LIN {X 0,Y 544.173,Z 839.846,A -85,B 0,C 180,E1 26201.66,E2 26201.66} C_VEL
LIN {X 0,Y 544.039,Z 847.664,A -85,B 0,C 180,E1 26199.734,E2 26199.734} C_VEL
LIN {X 0,Y 543.965,Z 854.535,A -85,B 0,C 180,E1 26197.605,E2 26197.605} C_VEL
LIN {X 0,Y 543.923,Z 859.536,A -85,B 0,C 180,E1 26195.485,E2 26195.485} C_VEL
LIN {X 0,Y 543.91,Z 862.863,A -85,B 0,C 180,E1 26193.445,E2 26193.445} C_VEL
LIN {X 0,Y 543.909,Z 864.729,A -85,B 0,C 180,E1 26191.159,E2 26191.159} C_VEL
LIN {X 0,Y 543.911,Z 864.816,A -85,B 0,C 180,E1 26189.157,E2 26189.157} C_VEL
LIN {X 0,Y 543.916,Z 863.417,A -85,B 0,C 180,E1 26187.05,E2 26187.05} C_VEL
LIN {X 0,Y 543.924,Z 860.152,A -85,B 0,C 180,E1 26184.832,E2 26184.832} C_VEL
LIN {X 0,Y 543.957,Z 855.674,A -85,B 0,C 180,E1 26182.82,E2 26182.82} C_VEL
LIN {X 0,Y 544.034,Z 848.851,A -85,B 0,C 180,E1 26180.586,E2 26180.586} C_VEL
LIN {X 0,Y 544.147,Z 841.239,A -85,B 0,C 180,E1 26178.662,E2 26178.662} C_VEL
LIN {X 0,Y 544.368,Z 831.448,A -85,B 0,C 180,E1 26176.619,E2 26176.619} C_VEL
LIN {X 0,Y 544.661,Z 820.069,A -85,B 0,C 180,E1 26174.672,E2 26174.672} C_VEL
LIN {X 0,Y 545.055,Z 807.802,A -85,B 0,C 180,E1 26172.89,E2 26172.89} C_VEL
LIN {X 0,Y 545.578,Z 792.93,A -85,B 0,C 180,E1 26171.073,E2 26171.073} C_VEL
LIN {X 0,Y 546.089,Z 779.11,A -85,B 0,C 180,E1 26169.629,E2 26169.629} C_VEL
LIN {X 0,Y 546.775,Z 762.015,A -85,B 0,C 180,E1 26168.097,E2 26168.097} C_VEL
LIN {X 0,Y 547.398,Z 745.705,A -85,B 0,C 180,E1 26166.877,E2 26166.877} C_VEL
LIN {X 0,Y 548.047,Z 728.308,A -85,B 0,C 180,E1 26165.765,E2 26165.765} C_VEL
LIN {X 0,Y 548.709,Z 708.264,A -85,B 0,C 180,E1 26164.73,E2 26164.73} C_VEL
LIN {X 0,Y 549.24,Z 690.742,A -85,B 0,C 180,E1 26164.006,E2 26164.006} C_VEL
LIN {X 0,Y 549.747,Z 670.512,A -85,B 0,C 180,E1 26163.357,E2 26163.357} C_VEL
LIN {X 0,Y 550.098,Z 650.393,A -85,B 0,C 180,E1 26162.921,E2 26162.921} C_VEL
LIN {X 0,Y 551.713,Z 417.884,A -85,B 0,C 180,E1 26159.601,E2 26159.601} C_VEL
LIN {X 0,Y 551.587,Z 408.026,A -85,B 0,C 180,E1 26159.447,E2 26159.447} C_VEL
LIN {X 0,Y 547.959,Z 394.771,A -85,B 0,C 180,E1 26158.998,E2 26158.998} C_VEL
LIN {X 0,Y 548.573,Z 372.146,A -85,B 0,C 180,E1 26156.171,E2 26156.171} C_VEL
LIN {X 0,Y 544.361,Z 357.302,A -85,B 0,C 180,E1 26153.906,E2 26153.906} C_VEL
LIN {X 0,Y 544.33,Z 357.175,A -85,B 0,C 180,E1 26150.489,E2 26150.489} C_VEL
LIN {X 0,Y 544.394,Z 357.168,A -85,B 0,C 180,E1 26147.281,E2 26147.281} C_VEL
LIN {X 0,Y 544.328,Z 357.176,A -85,B 0,C 180,E1 26144.094,E2 26144.094} C_VEL
LIN {X 0,Y 544.368,Z 357.177,A -85,B 0,C 180,E1 26140.825,E2 26140.825} C_VEL
LIN {X 0,Y 544.337,Z 357.171,A -85,B 0,C 180,E1 26137.713,E2 26137.713} C_VEL
LIN {X 0,Y 544.334,Z 357.172,A -85,B 0,C 180,E1 26134.329,E2 26134.329} C_VEL
LIN {X 0,Y 544.39,Z 357.175,A -85,B 0,C 180,E1 26131.074,E2 26131.074} C_VEL
LIN {X 0,Y 544.325,Z 357.163,A -85,B 0,C 180,E1 26127.815,E2 26127.815} C_VEL
LIN {X 0,Y 544.364,Z 357.176,A -85,B 0,C 180,E1 26124.529,E2 26124.529} C_VEL
LIN {X 0,Y 544.335,Z 357.165,A -85,B 0,C 180,E1 26121.444,E2 26121.444} C_VEL
LIN {X 0,Y 544.334,Z 357.177,A -85,B 0,C 180,E1 26118.088,E2 26118.088} C_VEL
LIN {X 0,Y 544.378,Z 357.166,A -85,B 0,C 180,E1 26114.904,E2 26114.904} C_VEL
LIN {X 0,Y 544.324,Z 357.175,A -85,B 0,C 180,E1 26111.661,E2 26111.661} C_VEL
LIN {X 0,Y 544.385,Z 357.169,A -85,B 0,C 180,E1 26108.453,E2 26108.453} C_VEL
LIN {X 0,Y 544.329,Z 357.166,A -85,B 0,C 180,E1 26105.274,E2 26105.274} C_VEL
LIN {X 0,Y 544.331,Z 357.176,A -85,B 0,C 180,E1 26101.794,E2 26101.794} C_VEL
LIN {X 0,Y 544.362,Z 357.164,A -85,B 0,C 180,E1 26098.742,E2 26098.742} C_VEL
LIN {X 0,Y 544.324,Z 357.175,A -85,B 0,C 180,E1 26095.475,E2 26095.475} C_VEL
LIN {X 0,Y 544.399,Z 357.166,A -85,B 0,C 180,E1 26092.3,E2 26092.3} C_VEL
LIN {X 0,Y 544.324,Z 357.169,A -85,B 0,C 180,E1 26089.099,E2 26089.099} C_VEL
LIN {X 0,Y 544.344,Z 357.175,A -85,B 0,C 180,E1 26085.757,E2 26085.757} C_VEL
LIN {X 0,Y 544.341,Z 357.162,A -85,B 0,C 180,E1 26082.695,E2 26082.695} C_VEL
LIN {X 0,Y 544.326,Z 357.177,A -85,B 0,C 180,E1 26079.355,E2 26079.355} C_VEL
LIN {X 0,Y 544.386,Z 357.164,A -85,B 0,C 180,E1 26076.154,E2 26076.154} C_VEL
LIN {X 0,Y 544.324,Z 357.177,A -85,B 0,C 180,E1 26072.907,E2 26072.907} C_VEL
LIN {X 0,Y 544.364,Z 357.177,A -85,B 0,C 180,E1 26069.669,E2 26069.669} C_VEL
LIN {X 0,Y 544.323,Z 357.177,A -85,B 0,C 180,E1 26069.105,E2 26069.105} C_VEL
LIN {X 0,Y 543.343,Z 357.304,A -85,B 0,C 180,E1 26068.295,E2 26068.295} C_VEL
LIN {X 0,Y 536.873,Z 358.114,A -85,B 0,C 180,E1 26065.958,E2 26065.958} C_VEL
LIN {X 0,Y 536.406,Z 358.167,A -85,B 0,C 180,E1 26065.424,E2 26065.424} C_VEL
LIN {X 0,Y 536.416,Z 358.165,A -85,B 0,C 180,E1 26062.213,E2 26062.213} C_VEL
LIN {X 0,Y 536.385,Z 358.167,A -85,B 0,C 180,E1 26059.003,E2 26059.003} C_VEL
LIN {X 0,Y 536.448,Z 358.166,A -85,B 0,C 180,E1 26055.817,E2 26055.817} C_VEL
LIN {X 0,Y 536.383,Z 358.167,A -85,B 0,C 180,E1 26052.582,E2 26052.582} C_VEL
LIN {X 0,Y 536.421,Z 358.166,A -85,B 0,C 180,E1 26049.325,E2 26049.325} C_VEL
LIN {X 0,Y 536.395,Z 358.167,A -85,B 0,C 180,E1 26046.197,E2 26046.197} C_VEL
LIN {X 0,Y 536.387,Z 358.167,A -85,B 0,C 180,E1 26042.802,E2 26042.802} C_VEL
LIN {X 0,Y 536.446,Z 358.165,A -85,B 0,C 180,E1 26039.598,E2 26039.598} C_VEL
LIN {X 0,Y 536.382,Z 358.167,A -85,B 0,C 180,E1 26036.336,E2 26036.336} C_VEL
LIN {X 0,Y 536.411,Z 358.167,A -85,B 0,C 180,E1 26032.978,E2 26032.978} C_VEL
LIN {X 0,Y 536.4,Z 358.166,A -85,B 0,C 180,E1 26029.831,E2 26029.831} C_VEL
LIN {X 0,Y 536.383,Z 358.168,A -85,B 0,C 180,E1 26026.459,E2 26026.459} C_VEL
LIN {X 0,Y 536.451,Z 358.165,A -85,B 0,C 180,E1 26023.253,E2 26023.253} C_VEL
LIN {X 0,Y 536.381,Z 358.167,A -85,B 0,C 180,E1 26019.983,E2 26019.983} C_VEL
LIN {X 0,Y 536.4,Z 358.168,A -85,B 0,C 180,E1 26016.602,E2 26016.602} C_VEL
LIN {X 0,Y 536.412,Z 358.166,A -85,B 0,C 180,E1 26013.419,E2 26013.419} C_VEL
LIN {X 0,Y 536.379,Z 358.168,A -85,B 0,C 180,E1 26010.107,E2 26010.107} C_VEL
LIN {X 0,Y 536.443,Z 358.168,A -85,B 0,C 180,E1 26006.902,E2 26006.902} C_VEL
LIN {X 0,Y 536.382,Z 358.168,A -85,B 0,C 180,E1 26003.686,E2 26003.686} C_VEL
LIN {X 0,Y 536.391,Z 358.167,A -85,B 0,C 180,E1 26000.234,E2 26000.234} C_VEL
LIN {X 0,Y 536.436,Z 358.166,A -85,B 0,C 180,E1 25996.966,E2 25996.966} C_VEL
LIN {X 0,Y 536.38,Z 358.168,A -85,B 0,C 180,E1 25993.71,E2 25993.71} C_VEL
LIN {X 0,Y 536.423,Z 358.166,A -85,B 0,C 180,E1 25990.397,E2 25990.397} C_VEL
LIN {X 0,Y 536.388,Z 358.167,A -85,B 0,C 180,E1 25987.303,E2 25987.303} C_VEL
LIN {X 0,Y 536.39,Z 358.167,A -85,B 0,C 180,E1 25983.902,E2 25983.902} C_VEL
LIN {X 0,Y 536.437,Z 358.166,A -85,B 0,C 180,E1 25980.71,E2 25980.71} C_VEL
LIN {X 0,Y 536.381,Z 358.167,A -85,B 0,C 180,E1 25977.531,E2 25977.531} C_VEL
LIN {X 0,Y 536.442,Z 358.167,A -85,B 0,C 180,E1 25974.312,E2 25974.312} C_VEL
LIN {X 0,Y 536.388,Z 358.166,A -85,B 0,C 180,E1 25971.085,E2 25971.085} C_VEL
LIN {X 0,Y 536.387,Z 358.167,A -85,B 0,C 180,E1 25967.564,E2 25967.564} C_VEL
LIN {X 0,Y 536.45,Z 358.165,A -85,B 0,C 180,E1 25964.3,E2 25964.3} C_VEL
LIN {X 0,Y 536.382,Z 358.167,A -85,B 0,C 180,E1 25961.139,E2 25961.139} C_VEL
LIN {X 0,Y 536.42,Z 358.165,A -85,B 0,C 180,E1 25957.815,E2 25957.815} C_VEL
LIN {X 0,Y 536.401,Z 358.167,A -85,B 0,C 180,E1 25954.639,E2 25954.639} C_VEL
LIN {X 0,Y 536.389,Z 358.166,A -85,B 0,C 180,E1 25951.329,E2 25951.329} C_VEL
LIN {X 0,Y 536.446,Z 358.166,A -85,B 0,C 180,E1 25948.128,E2 25948.128} C_VEL
LIN {X 0,Y 536.382,Z 358.158,A -85,B 0,C 180,E1 25944.908,E2 25944.908} C_VEL
LIN {X 0,Y 536.433,Z 358.165,A -85,B 0,C 180,E1 25941.651,E2 25941.651} C_VEL
LIN {X 0,Y 536.399,Z 358.162,A -85,B 0,C 180,E1 25938.421,E2 25938.421} C_VEL
LIN {X 0,Y 536.386,Z 358.163,A -85,B 0,C 180,E1 25935.011,E2 25935.011} C_VEL
LIN {X 0,Y 536.449,Z 358.161,A -85,B 0,C 180,E1 25931.825,E2 25931.825} C_VEL
LIN {X 0,Y 536.383,Z 358.153,A -85,B 0,C 180,E1 25928.571,E2 25928.571} C_VEL
LIN {X 0,Y 536.428,Z 358.164,A -85,B 0,C 180,E1 25925.342,E2 25925.342} C_VEL
LIN {X 0,Y 536.4,Z 358.155,A -85,B 0,C 180,E1 25922.132,E2 25922.132} C_VEL
LIN {X 0,Y 536.388,Z 358.164,A -85,B 0,C 180,E1 25918.714,E2 25918.714} C_VEL
LIN {X 0,Y 536.451,Z 358.156,A -85,B 0,C 180,E1 25915.506,E2 25915.506} C_VEL
LIN {X 0,Y 536.385,Z 358.156,A -85,B 0,C 180,E1 25912.283,E2 25912.283} C_VEL
LIN {X 0,Y 536.413,Z 358.163,A -85,B 0,C 180,E1 25908.927,E2 25908.927} C_VEL
LIN {X 0,Y 536.411,Z 358.151,A -85,B 0,C 180,E1 25905.752,E2 25905.752} C_VEL
LIN {X 0,Y 536.388,Z 358.165,A -85,B 0,C 180,E1 25902.42,E2 25902.42} C_VEL
LIN {X 0,Y 536.455,Z 358.149,A -85,B 0,C 180,E1 25899.142,E2 25899.142} C_VEL
LIN {X 0,Y 536.391,Z 358.165,A -85,B 0,C 180,E1 25895.903,E2 25895.903} C_VEL
LIN {X 0,Y 536.399,Z 358.15,A -85,B 0,C 180,E1 25892.463,E2 25892.463} C_VEL
LIN {X 0,Y 536.442,Z 358.165,A -85,B 0,C 180,E1 25889.229,E2 25889.229} C_VEL
LIN {X 0,Y 536.387,Z 358.161,A -85,B 0,C 180,E1 25885.995,E2 25885.995} C_VEL
LIN {X 0,Y 536.438,Z 358.157,A -85,B 0,C 180,E1 25882.714,E2 25882.714} C_VEL
LIN {X 0,Y 536.396,Z 358.167,A -85,B 0,C 180,E1 25879.555,E2 25879.555} C_VEL
LIN {X 0,Y 536.395,Z 358.165,A -85,B 0,C 180,E1 25876.096,E2 25876.096} C_VEL
LIN {X 0,Y 536.453,Z 358.159,A -85,B 0,C 180,E1 25872.865,E2 25872.865} C_VEL
LIN {X 0,Y 536.389,Z 358.161,A -85,B 0,C 180,E1 25869.605,E2 25869.605} C_VEL
LIN {X 0,Y 536.475,Z 358.365,A -85,B 0,C 180,E1 25866.512,E2 25866.512} C_VEL
LIN {X 0,Y 541.121,Z 374.813,A -85,B 0,C 180,E1 25863.975,E2 25863.975} C_VEL
LIN {X 0,Y 540.557,Z 394.905,A -85,B 0,C 180,E1 25861.456,E2 25861.456} C_VEL
LIN {X 0,Y 544.864,Z 411.254,A -85,B 0,C 180,E1 25860.922,E2 25860.922} C_VEL
LIN {X 0,Y 543.047,Z 645.18,A -85,B 0,C 180,E1 25857.554,E2 25857.554} C_VEL
LIN {X 0,Y 542.717,Z 664.023,A -85,B 0,C 180,E1 25857.181,E2 25857.181} C_VEL
LIN {X 0,Y 542.237,Z 682.867,A -85,B 0,C 180,E1 25856.649,E2 25856.649} C_VEL
LIN {X 0,Y 541.576,Z 703.966,A -85,B 0,C 180,E1 25855.829,E2 25855.829} C_VEL
LIN {X 0,Y 540.927,Z 721.195,A -85,B 0,C 180,E1 25854.983,E2 25854.983} C_VEL
LIN {X 0,Y 540.186,Z 739.996,A -85,B 0,C 180,E1 25853.861,E2 25853.861} C_VEL
LIN {X 0,Y 539.423,Z 757.066,A -85,B 0,C 180,E1 25852.618,E2 25852.618} C_VEL
LIN {X 0,Y 538.693,Z 773.48,A -85,B 0,C 180,E1 25851.218,E2 25851.218} C_VEL
LIN {X 0,Y 537.963,Z 789.942,A -85,B 0,C 180,E1 25849.544,E2 25849.544} C_VEL
LIN {X 0,Y 537.382,Z 803.934,A -85,B 0,C 180,E1 25847.878,E2 25847.878} C_VEL
LIN {X 0,Y 536.859,Z 817.974,A -85,B 0,C 180,E1 25845.889,E2 25845.889} C_VEL
LIN {X 0,Y 536.503,Z 829.096,A -85,B 0,C 180,E1 25844.02,E2 25844.02} C_VEL
LIN {X 0,Y 536.212,Z 839.843,A -85,B 0,C 180,E1 25841.836,E2 25841.836} C_VEL
LIN {X 0,Y 536.058,Z 847.659,A -85,B 0,C 180,E1 25839.88,E2 25839.88} C_VEL
LIN {X 0,Y 535.974,Z 854.538,A -85,B 0,C 180,E1 25837.719,E2 25837.719} C_VEL
LIN {X 0,Y 535.926,Z 859.534,A -85,B 0,C 180,E1 25835.567,E2 25835.567} C_VEL
LIN {X 0,Y 535.91,Z 862.897,A -85,B 0,C 180,E1 25833.468,E2 25833.468} C_VEL
LIN {X 0,Y 535.908,Z 864.725,A -85,B 0,C 180,E1 25831.176,E2 25831.176} C_VEL
LIN {X 0,Y 535.911,Z 864.812,A -85,B 0,C 180,E1 25829.145,E2 25829.145} C_VEL
LIN {X 0,Y 535.915,Z 863.42,A -85,B 0,C 180,E1 25827.006,E2 25827.006} C_VEL
LIN {X 0,Y 535.924,Z 860.15,A -85,B 0,C 180,E1 25824.755,E2 25824.755} C_VEL
LIN {X 0,Y 535.962,Z 855.669,A -85,B 0,C 180,E1 25822.712,E2 25822.712} C_VEL
LIN {X 0,Y 536.051,Z 848.846,A -85,B 0,C 180,E1 25820.445,E2 25820.445} C_VEL
LIN {X 0,Y 536.187,Z 841.236,A -85,B 0,C 180,E1 25818.491,E2 25818.491} C_VEL
LIN {X 0,Y 536.444,Z 831.453,A -85,B 0,C 180,E1 25816.418,E2 25816.418} C_VEL
LIN {X 0,Y 536.784,Z 820.064,A -85,B 0,C 180,E1 25814.442,E2 25814.442} C_VEL
LIN {X 0,Y 537.226,Z 808.102,A -85,B 0,C 180,E1 25812.676,E2 25812.676} C_VEL
LIN {X 0,Y 537.833,Z 793.069,A -85,B 0,C 180,E1 25810.806,E2 25810.806} C_VEL
LIN {X 0,Y 538.42,Z 779.248,A -85,B 0,C 180,E1 25809.34,E2 25809.34} C_VEL
LIN {X 0,Y 539.205,Z 762.007,A -85,B 0,C 180,E1 25807.773,E2 25807.773} C_VEL
LIN {X 0,Y 539.916,Z 745.7,A -85,B 0,C 180,E1 25806.538,E2 25806.538} C_VEL
LIN {X 0,Y 540.61,Z 729.214,A -85,B 0,C 180,E1 25805.468,E2 25805.468} C_VEL
LIN {X 0,Y 541.383,Z 708.932,A -85,B 0,C 180,E1 25804.396,E2 25804.396} C_VEL
LIN {X 0,Y 541.969,Z 691.817,A -85,B 0,C 180,E1 25803.674,E2 25803.674} C_VEL
LIN {X 0,Y 542.539,Z 672.217,A -85,B 0,C 180,E1 25803.023,E2 25803.023} C_VEL
LIN {X 0,Y 542.957,Z 651.512,A -85,B 0,C 180,E1 25802.556,E2 25802.556} C_VEL
LIN {X 0,Y 544.781,Z 422.259,A -85,B 0,C 180,E1 25799.238,E2 25799.238} C_VEL
LIN {X 0,Y 544.663,Z 409.644,A -85,B 0,C 180,E1 25799.041,E2 25799.041} C_VEL
LIN {X 0,Y 540.517,Z 394.526,A -85,B 0,C 180,E1 25798.516,E2 25798.516} C_VEL
LIN {X 0,Y 541.014,Z 374.271,A -85,B 0,C 180,E1 25795.947,E2 25795.947} C_VEL
LIN {X 0,Y 536.462,Z 358.25,A -85,B 0,C 180,E1 25793.448,E2 25793.448} C_VEL
LIN {X 0,Y 536.388,Z 358.156,A -85,B 0,C 180,E1 25790.176,E2 25790.176} C_VEL
LIN {X 0,Y 536.421,Z 358.169,A -85,B 0,C 180,E1 25786.839,E2 25786.839} C_VEL
LIN {X 0,Y 536.415,Z 358.164,A -85,B 0,C 180,E1 25783.606,E2 25783.606} C_VEL
LIN {X 0,Y 536.391,Z 358.167,A -85,B 0,C 180,E1 25780.305,E2 25780.305} C_VEL
LIN {X 0,Y 536.456,Z 358.157,A -85,B 0,C 180,E1 25777.09,E2 25777.09} C_VEL
LIN {X 0,Y 536.39,Z 358.16,A -85,B 0,C 180,E1 25773.876,E2 25773.876} C_VEL
LIN {X 0,Y 536.417,Z 358.165,A -85,B 0,C 180,E1 25770.557,E2 25770.557} C_VEL
LIN {X 0,Y 536.407,Z 358.15,A -85,B 0,C 180,E1 25767.416,E2 25767.416} C_VEL
LIN {X 0,Y 536.389,Z 358.165,A -85,B 0,C 180,E1 25764.026,E2 25764.026} C_VEL
LIN {X 0,Y 536.455,Z 358.149,A -85,B 0,C 180,E1 25760.858,E2 25760.858} C_VEL
LIN {X 0,Y 536.388,Z 358.165,A -85,B 0,C 180,E1 25757.58,E2 25757.58} C_VEL
LIN {X 0,Y 536.411,Z 358.151,A -85,B 0,C 180,E1 25754.247,E2 25754.247} C_VEL
LIN {X 0,Y 536.413,Z 358.163,A -85,B 0,C 180,E1 25751.073,E2 25751.073} C_VEL
LIN {X 0,Y 536.385,Z 358.156,A -85,B 0,C 180,E1 25747.717,E2 25747.717} C_VEL
LIN {X 0,Y 536.451,Z 358.156,A -85,B 0,C 180,E1 25744.494,E2 25744.494} C_VEL
LIN {X 0,Y 536.388,Z 358.164,A -85,B 0,C 180,E1 25741.286,E2 25741.286} C_VEL
LIN {X 0,Y 536.4,Z 358.155,A -85,B 0,C 180,E1 25737.868,E2 25737.868} C_VEL
LIN {X 0,Y 536.428,Z 358.164,A -85,B 0,C 180,E1 25734.658,E2 25734.658} C_VEL
LIN {X 0,Y 536.383,Z 358.153,A -85,B 0,C 180,E1 25731.429,E2 25731.429} C_VEL
LIN {X 0,Y 536.449,Z 358.161,A -85,B 0,C 180,E1 25728.175,E2 25728.175} C_VEL
LIN {X 0,Y 536.386,Z 358.163,A -85,B 0,C 180,E1 25724.989,E2 25724.989} C_VEL
LIN {X 0,Y 536.395,Z 358.162,A -85,B 0,C 180,E1 25721.532,E2 25721.532} C_VEL
LIN {X 0,Y 536.433,Z 358.165,A -85,B 0,C 180,E1 25718.349,E2 25718.349} C_VEL
LIN {X 0,Y 536.382,Z 358.158,A -85,B 0,C 180,E1 25715.092,E2 25715.092} C_VEL
LIN {X 0,Y 536.441,Z 358.166,A -85,B 0,C 180,E1 25711.834,E2 25711.834} C_VEL
LIN {X 0,Y 536.389,Z 358.166,A -85,B 0,C 180,E1 25708.671,E2 25708.671} C_VEL
LIN {X 0,Y 536.406,Z 358.167,A -85,B 0,C 180,E1 25705.424,E2 25705.424} C_VEL
LIN {X 0,Y 535.4,Z 358.29,A -85,B 0,C 180,E1 25704.602,E2 25704.602} C_VEL
LIN {X 0,Y 528.983,Z 359.1,A -85,B 0,C 180,E1 25702.231,E2 25702.231} C_VEL
LIN {X 0,Y 528.504,Z 359.154,A -85,B 0,C 180,E1 25701.689,E2 25701.689} C_VEL
LIN {X 0,Y 528.449,Z 359.155,A -85,B 0,C 180,E1 25698.524,E2 25698.524} C_VEL
LIN {X 0,Y 528.451,Z 359.156,A -85,B 0,C 180,E1 25695.041,E2 25695.041} C_VEL
LIN {X 0,Y 528.51,Z 359.154,A -85,B 0,C 180,E1 25691.752,E2 25691.752} C_VEL
LIN {X 0,Y 528.445,Z 359.155,A -85,B 0,C 180,E1 25688.447,E2 25688.447} C_VEL
LIN {X 0,Y 528.456,Z 359.156,A -85,B 0,C 180,E1 25684.979,E2 25684.979} C_VEL
LIN {X 0,Y 528.493,Z 359.155,A -85,B 0,C 180,E1 25681.731,E2 25681.731} C_VEL
LIN {X 0,Y 528.444,Z 359.155,A -85,B 0,C 180,E1 25678.476,E2 25678.476} C_VEL
LIN {X 0,Y 528.493,Z 359.156,A -85,B 0,C 180,E1 25675.193,E2 25675.193} C_VEL
LIN {X 0,Y 528.451,Z 359.156,A -85,B 0,C 180,E1 25672.001,E2 25672.001} C_VEL
LIN {X 0,Y 528.446,Z 359.156,A -85,B 0,C 180,E1 25668.533,E2 25668.533} C_VEL
LIN {X 0,Y 528.515,Z 359.153,A -85,B 0,C 180,E1 25665.246,E2 25665.246} C_VEL
LIN {X 0,Y 528.443,Z 359.155,A -85,B 0,C 180,E1 25662.012,E2 25662.012} C_VEL
LIN {X 0,Y 528.458,Z 359.157,A -85,B 0,C 180,E1 25658.596,E2 25658.596} C_VEL
LIN {X 0,Y 528.476,Z 359.156,A -85,B 0,C 180,E1 25655.428,E2 25655.428} C_VEL
LIN {X 0,Y 528.439,Z 359.157,A -85,B 0,C 180,E1 25652.06,E2 25652.06} C_VEL
LIN {X 0,Y 528.495,Z 359.157,A -85,B 0,C 180,E1 25648.808,E2 25648.808} C_VEL
LIN {X 0,Y 528.453,Z 359.155,A -85,B 0,C 180,E1 25645.527,E2 25645.527} C_VEL
LIN {X 0,Y 528.448,Z 359.157,A -85,B 0,C 180,E1 25642.171,E2 25642.171} C_VEL
LIN {X 0,Y 528.497,Z 359.155,A -85,B 0,C 180,E1 25638.984,E2 25638.984} C_VEL
LIN {X 0,Y 528.44,Z 359.157,A -85,B 0,C 180,E1 25635.761,E2 25635.761} C_VEL
LIN {X 0,Y 528.485,Z 359.156,A -85,B 0,C 180,E1 25632.436,E2 25632.436} C_VEL
LIN {X 0,Y 528.453,Z 359.155,A -85,B 0,C 180,E1 25629.28,E2 25629.28} C_VEL
LIN {X 0,Y 528.448,Z 359.157,A -85,B 0,C 180,E1 25625.878,E2 25625.878} C_VEL
LIN {X 0,Y 528.516,Z 359.154,A -85,B 0,C 180,E1 25622.513,E2 25622.513} C_VEL
LIN {X 0,Y 528.445,Z 359.156,A -85,B 0,C 180,E1 25619.28,E2 25619.28} C_VEL
LIN {X 0,Y 528.454,Z 359.156,A -85,B 0,C 180,E1 25615.811,E2 25615.811} C_VEL
LIN {X 0,Y 528.492,Z 359.155,A -85,B 0,C 180,E1 25612.604,E2 25612.604} C_VEL
LIN {X 0,Y 528.442,Z 359.155,A -85,B 0,C 180,E1 25609.34,E2 25609.34} C_VEL
LIN {X 0,Y 528.491,Z 359.156,A -85,B 0,C 180,E1 25606.028,E2 25606.028} C_VEL
LIN {X 0,Y 528.461,Z 359.156,A -85,B 0,C 180,E1 25602.77,E2 25602.77} C_VEL
LIN {X 0,Y 528.45,Z 359.155,A -85,B 0,C 180,E1 25599.465,E2 25599.465} C_VEL
LIN {X 0,Y 528.498,Z 359.155,A -85,B 0,C 180,E1 25596.301,E2 25596.301} C_VEL
LIN {X 0,Y 528.445,Z 359.156,A -85,B 0,C 180,E1 25593.011,E2 25593.011} C_VEL
LIN {X 0,Y 528.484,Z 359.155,A -85,B 0,C 180,E1 25589.707,E2 25589.707} C_VEL
LIN {X 0,Y 528.463,Z 359.155,A -85,B 0,C 180,E1 25586.505,E2 25586.505} C_VEL
LIN {X 0,Y 528.449,Z 359.147,A -85,B 0,C 180,E1 25583.145,E2 25583.145} C_VEL
LIN {X 0,Y 528.512,Z 359.153,A -85,B 0,C 180,E1 25579.903,E2 25579.903} C_VEL
LIN {X 0,Y 528.447,Z 359.138,A -85,B 0,C 180,E1 25576.595,E2 25576.595} C_VEL
LIN {X 0,Y 528.456,Z 359.154,A -85,B 0,C 180,E1 25573.117,E2 25573.117} C_VEL
LIN {X 0,Y 528.495,Z 359.138,A -85,B 0,C 180,E1 25569.908,E2 25569.908} C_VEL
LIN {X 0,Y 528.445,Z 359.153,A -85,B 0,C 180,E1 25566.622,E2 25566.622} C_VEL
LIN {X 0,Y 528.492,Z 359.142,A -85,B 0,C 180,E1 25563.357,E2 25563.357} C_VEL
LIN {X 0,Y 528.46,Z 359.143,A -85,B 0,C 180,E1 25560.104,E2 25560.104} C_VEL
LIN {X 0,Y 528.452,Z 359.153,A -85,B 0,C 180,E1 25556.742,E2 25556.742} C_VEL
LIN {X 0,Y 528.516,Z 359.134,A -85,B 0,C 180,E1 25553.478,E2 25553.478} C_VEL
LIN {X 0,Y 528.45,Z 359.154,A -85,B 0,C 180,E1 25550.192,E2 25550.192} C_VEL
LIN {X 0,Y 528.461,Z 359.139,A -85,B 0,C 180,E1 25546.762,E2 25546.762} C_VEL
LIN {X 0,Y 528.482,Z 359.148,A -85,B 0,C 180,E1 25543.623,E2 25543.623} C_VEL
LIN {X 0,Y 528.448,Z 359.149,A -85,B 0,C 180,E1 25540.315,E2 25540.315} C_VEL
LIN {X 0,Y 528.512,Z 359.147,A -85,B 0,C 180,E1 25537.06,E2 25537.06} C_VEL
LIN {X 0,Y 528.455,Z 359.153,A -85,B 0,C 180,E1 25533.839,E2 25533.839} C_VEL
LIN {X 0,Y 528.459,Z 359.153,A -85,B 0,C 180,E1 25530.405,E2 25530.405} C_VEL
LIN {X 0,Y 528.497,Z 359.148,A -85,B 0,C 180,E1 25527.24,E2 25527.24} C_VEL
LIN {X 0,Y 528.449,Z 359.155,A -85,B 0,C 180,E1 25523.951,E2 25523.951} C_VEL
LIN {X 0,Y 528.499,Z 359.155,A -85,B 0,C 180,E1 25520.668,E2 25520.668} C_VEL
LIN {X 0,Y 528.459,Z 359.153,A -85,B 0,C 180,E1 25517.508,E2 25517.508} C_VEL
LIN {X 0,Y 528.455,Z 359.158,A -85,B 0,C 180,E1 25514.028,E2 25514.028} C_VEL
LIN {X 0,Y 528.519,Z 359.123,A -85,B 0,C 180,E1 25510.742,E2 25510.742} C_VEL
LIN {X 0,Y 528.45,Z 359.136,A -85,B 0,C 180,E1 25507.533,E2 25507.533} C_VEL
LIN {X 0,Y 528.547,Z 359.504,A -85,B 0,C 180,E1 25506.943,E2 25506.943} C_VEL
LIN {X 0,Y 533.673,Z 377.481,A -85,B 0,C 180,E1 25504.126,E2 25504.126} C_VEL
LIN {X 0,Y 533.115,Z 394.665,A -85,B 0,C 180,E1 25501.944,E2 25501.944} C_VEL
LIN {X 0,Y 537.976,Z 412.936,A -85,B 0,C 180,E1 25501.334,E2 25501.334} C_VEL
LIN {X 0,Y 535.952,Z 645.248,A -85,B 0,C 180,E1 25497.949,E2 25497.949} C_VEL
LIN {X 0,Y 535.585,Z 663.92,A -85,B 0,C 180,E1 25497.575,E2 25497.575} C_VEL
LIN {X 0,Y 535.084,Z 681.927,A -85,B 0,C 180,E1 25497.064,E2 25497.064} C_VEL
LIN {X 0,Y 534.375,Z 702.71,A -85,B 0,C 180,E1 25496.263,E2 25496.263} C_VEL
LIN {X 0,Y 533.656,Z 719.661,A -85,B 0,C 180,E1 25495.432,E2 25495.432} C_VEL
LIN {X 0,Y 532.875,Z 737.458,A -85,B 0,C 180,E1 25494.38,E2 25494.38} C_VEL
LIN {X 0,Y 531.97,Z 755.622,A -85,B 0,C 180,E1 25493.071,E2 25493.071} C_VEL
LIN {X 0,Y 531.17,Z 771.475,A -85,B 0,C 180,E1 25491.72,E2 25491.72} C_VEL
LIN {X 0,Y 530.317,Z 788.658,A -85,B 0,C 180,E1 25489.986,E2 25489.986} C_VEL
LIN {X 0,Y 529.68,Z 802.156,A -85,B 0,C 180,E1 25488.375,E2 25488.375} C_VEL
LIN {X 0,Y 529.096,Z 815.857,A -85,B 0,C 180,E1 25486.466,E2 25486.466} C_VEL
LIN {X 0,Y 528.65,Z 827.248,A -85,B 0,C 180,E1 25484.569,E2 25484.569} C_VEL
LIN {X 0,Y 528.337,Z 837.389,A -85,B 0,C 180,E1 25482.57,E2 25482.57} C_VEL
LIN {X 0,Y 528.111,Z 846.468,A -85,B 0,C 180,E1 25480.361,E2 25480.361} C_VEL
LIN {X 0,Y 528.002,Z 853.31,A -85,B 0,C 180,E1 25478.274,E2 25478.274} C_VEL
LIN {X 0,Y 527.937,Z 858.915,A -85,B 0,C 180,E1 25475.979,E2 25475.979} C_VEL
LIN {X 0,Y 527.916,Z 862.371,A -85,B 0,C 180,E1 25473.91,E2 25473.91} C_VEL
LIN {X 0,Y 527.907,Z 864.467,A -85,B 0,C 180,E1 25471.737,E2 25471.737} C_VEL
LIN {X 0,Y 527.9,Z 864.895,A -85,B 0,C 180,E1 25469.457,E2 25469.457} C_VEL
LIN {X 0,Y 527.908,Z 863.727,A -85,B 0,C 180,E1 25467.286,E2 25467.286} C_VEL
LIN {X 0,Y 527.928,Z 860.763,A -85,B 0,C 180,E1 25465.002,E2 25465.002} C_VEL
LIN {X 0,Y 527.963,Z 856.429,A -85,B 0,C 180,E1 25462.915,E2 25462.915} C_VEL
LIN {X 0,Y 528.047,Z 850.301,A -85,B 0,C 180,E1 25460.738,E2 25460.738} C_VEL
LIN {X 0,Y 528.208,Z 842.161,A -85,B 0,C 180,E1 25458.536,E2 25458.536} C_VEL
LIN {X 0,Y 528.445,Z 833.662,A -85,B 0,C 180,E1 25456.654,E2 25456.654} C_VEL
LIN {X 0,Y 528.841,Z 822.149,A -85,B 0,C 180,E1 25454.539,E2 25454.539} C_VEL
LIN {X 0,Y 529.302,Z 810.456,A -85,B 0,C 180,E1 25452.749,E2 25452.749} C_VEL
LIN {X 0,Y 529.935,Z 796.797,A -85,B 0,C 180,E1 25450.95,E2 25450.95} C_VEL
LIN {X 0,Y 530.658,Z 781.474,A -85,B 0,C 180,E1 25449.255,E2 25449.255} C_VEL
LIN {X 0,Y 531.462,Z 765.955,A -85,B 0,C 180,E1 25447.782,E2 25447.782} C_VEL
LIN {X 0,Y 532.348,Z 748.104,A -85,B 0,C 180,E1 25446.36,E2 25446.36} C_VEL
LIN {X 0,Y 533.093,Z 731.955,A -85,B 0,C 180,E1 25445.276,E2 25445.276} C_VEL
LIN {X 0,Y 533.967,Z 713.091,A -85,B 0,C 180,E1 25444.218,E2 25444.218} C_VEL
LIN {X 0,Y 534.689,Z 693.683,A -85,B 0,C 180,E1 25443.363,E2 25443.363} C_VEL
LIN {X 0,Y 535.243,Z 676.556,A -85,B 0,C 180,E1 25442.768,E2 25442.768} C_VEL
LIN {X 0,Y 535.797,Z 655.919,A -85,B 0,C 180,E1 25442.239,E2 25442.239} C_VEL
LIN {X 0,Y 536.204,Z 618.298,A -85,B 0,C 180,E1 25441.656,E2 25441.656} C_VEL
LIN {X 0,Y 537.913,Z 411.946,A -85,B 0,C 180,E1 25438.647,E2 25438.647} C_VEL
LIN {X 0,Y 533.079,Z 394.366,A -85,B 0,C 180,E1 25438.036,E2 25438.036} C_VEL
LIN {X 0,Y 533.561,Z 376.939,A -85,B 0,C 180,E1 25435.794,E2 25435.794} C_VEL
LIN {X 0,Y 528.5,Z 359.245,A -85,B 0,C 180,E1 25432.997,E2 25432.997} C_VEL
LIN {X 0,Y 528.465,Z 359.134,A -85,B 0,C 180,E1 25429.823,E2 25429.823} C_VEL
LIN {X 0,Y 528.456,Z 359.158,A -85,B 0,C 180,E1 25426.442,E2 25426.442} C_VEL
LIN {X 0,Y 528.516,Z 359.154,A -85,B 0,C 180,E1 25423.226,E2 25423.226} C_VEL
LIN {X 0,Y 528.452,Z 359.155,A -85,B 0,C 180,E1 25419.981,E2 25419.981} C_VEL
LIN {X 0,Y 528.48,Z 359.156,A -85,B 0,C 180,E1 25416.663,E2 25416.663} C_VEL
LIN {X 0,Y 528.474,Z 359.148,A -85,B 0,C 180,E1 25413.453,E2 25413.453} C_VEL
LIN {X 0,Y 528.451,Z 359.153,A -85,B 0,C 180,E1 25410.095,E2 25410.095} C_VEL
LIN {X 0,Y 528.514,Z 359.14,A -85,B 0,C 180,E1 25406.885,E2 25406.885} C_VEL
LIN {X 0,Y 528.451,Z 359.153,A -85,B 0,C 180,E1 25403.651,E2 25403.651} C_VEL
LIN {X 0,Y 528.462,Z 359.15,A -85,B 0,C 180,E1 25400.214,E2 25400.214} C_VEL
LIN {X 0,Y 528.485,Z 359.154,A -85,B 0,C 180,E1 25397.056,E2 25397.056} C_VEL
LIN {X 0,Y 528.447,Z 359.14,A -85,B 0,C 180,E1 25393.796,E2 25393.796} C_VEL
LIN {X 0,Y 528.502,Z 359.155,A -85,B 0,C 180,E1 25390.468,E2 25390.468} C_VEL
LIN {X 0,Y 528.453,Z 359.144,A -85,B 0,C 180,E1 25387.287,E2 25387.287} C_VEL
LIN {X 0,Y 528.453,Z 359.153,A -85,B 0,C 180,E1 25383.801,E2 25383.801} C_VEL
LIN {X 0,Y 528.52,Z 359.143,A -85,B 0,C 180,E1 25380.438,E2 25380.438} C_VEL
LIN {X 0,Y 528.449,Z 359.143,A -85,B 0,C 180,E1 25377.185,E2 25377.185} C_VEL
LIN {X 0,Y 528.455,Z 359.153,A -85,B 0,C 180,E1 25373.705,E2 25373.705} C_VEL
LIN {X 0,Y 528.493,Z 359.136,A -85,B 0,C 180,E1 25370.532,E2 25370.532} C_VEL
LIN {X 0,Y 528.445,Z 359.155,A -85,B 0,C 180,E1 25367.216,E2 25367.216} C_VEL
LIN {X 0,Y 528.491,Z 359.138,A -85,B 0,C 180,E1 25363.958,E2 25363.958} C_VEL
LIN {X 0,Y 528.463,Z 359.15,A -85,B 0,C 180,E1 25360.671,E2 25360.671} C_VEL
LIN {X 0,Y 528.448,Z 359.147,A -85,B 0,C 180,E1 25357.302,E2 25357.302} C_VEL
LIN {X 0,Y 528.509,Z 359.149,A -85,B 0,C 180,E1 25353.973,E2 25353.973} C_VEL
LIN {X 0,Y 528.45,Z 359.155,A -85,B 0,C 180,E1 25350.717,E2 25350.717} C_VEL
LIN {X 0,Y 528.453,Z 359.156,A -85,B 0,C 180,E1 25347.248,E2 25347.248} C_VEL
LIN {X 0,Y 528.508,Z 359.155,A -85,B 0,C 180,E1 25343.968,E2 25343.968} C_VEL
LIN {X 0,Y 528.504,Z 359.154,A -85,B 0,C 180,E1 25341.689,E2 25341.689} C_VEL
LIN {X 0,Y 527.438,Z 359.283,A -85,B 0,C 180,E1 25340.854,E2 25340.854} C_VEL
LIN {X 0,Y 521.043,Z 360.085,A -85,B 0,C 180,E1 25338.509,E2 25338.509} C_VEL
LIN {X 0,Y 520.565,Z 360.144,A -85,B 0,C 180,E1 25337.898,E2 25337.898} C_VEL
LIN {X 0,Y 520.508,Z 360.145,A -85,B 0,C 180,E1 25334.559,E2 25334.559} C_VEL
LIN {X 0,Y 520.517,Z 360.144,A -85,B 0,C 180,E1 25331.066,E2 25331.066} C_VEL
LIN {X 0,Y 520.548,Z 360.144,A -85,B 0,C 180,E1 25327.88,E2 25327.88} C_VEL
LIN {X 0,Y 520.504,Z 360.145,A -85,B 0,C 180,E1 25324.518,E2 25324.518} C_VEL
LIN {X 0,Y 520.547,Z 360.145,A -85,B 0,C 180,E1 25321.238,E2 25321.238} C_VEL
LIN {X 0,Y 520.516,Z 360.144,A -85,B 0,C 180,E1 25318.074,E2 25318.074} C_VEL
LIN {X 0,Y 520.507,Z 360.146,A -85,B 0,C 180,E1 25314.635,E2 25314.635} C_VEL
LIN {X 0,Y 520.573,Z 360.143,A -85,B 0,C 180,E1 25311.349,E2 25311.349} C_VEL
LIN {X 0,Y 520.509,Z 360.146,A -85,B 0,C 180,E1 25308.015,E2 25308.015} C_VEL
LIN {X 0,Y 520.507,Z 360.146,A -85,B 0,C 180,E1 25304.461,E2 25304.461} C_VEL
LIN {X 0,Y 520.566,Z 360.145,A -85,B 0,C 180,E1 25301.186,E2 25301.186} C_VEL
LIN {X 0,Y 520.503,Z 360.146,A -85,B 0,C 180,E1 25297.95,E2 25297.95} C_VEL
LIN {X 0,Y 520.517,Z 360.145,A -85,B 0,C 180,E1 25294.517,E2 25294.517} C_VEL
LIN {X 0,Y 520.553,Z 360.146,A -85,B 0,C 180,E1 25291.211,E2 25291.211} C_VEL
LIN {X 0,Y 520.501,Z 360.146,A -85,B 0,C 180,E1 25287.908,E2 25287.908} C_VEL
LIN {X 0,Y 520.529,Z 360.146,A -85,B 0,C 180,E1 25284.489,E2 25284.489} C_VEL
LIN {X 0,Y 520.521,Z 360.146,A -85,B 0,C 180,E1 25281.383,E2 25281.383} C_VEL
LIN {X 0,Y 520.506,Z 360.144,A -85,B 0,C 180,E1 25278.027,E2 25278.027} C_VEL
LIN {X 0,Y 520.575,Z 360.142,A -85,B 0,C 180,E1 25274.744,E2 25274.744} C_VEL
LIN {X 0,Y 520.51,Z 360.146,A -85,B 0,C 180,E1 25271.406,E2 25271.406} C_VEL
LIN {X 0,Y 520.509,Z 360.145,A -85,B 0,C 180,E1 25267.884,E2 25267.884} C_VEL
LIN {X 0,Y 520.567,Z 360.143,A -85,B 0,C 180,E1 25264.64,E2 25264.64} C_VEL
LIN {X 0,Y 520.505,Z 360.145,A -85,B 0,C 180,E1 25261.369,E2 25261.369} C_VEL
LIN {X 0,Y 520.526,Z 360.145,A -85,B 0,C 180,E1 25257.985,E2 25257.985} C_VEL
LIN {X 0,Y 520.549,Z 360.145,A -85,B 0,C 180,E1 25254.68,E2 25254.68} C_VEL
LIN {X 0,Y 520.503,Z 360.144,A -85,B 0,C 180,E1 25251.37,E2 25251.37} C_VEL
LIN {X 0,Y 520.549,Z 360.144,A -85,B 0,C 180,E1 25248.056,E2 25248.056} C_VEL
LIN {X 0,Y 520.522,Z 360.145,A -85,B 0,C 180,E1 25244.816,E2 25244.816} C_VEL
LIN {X 0,Y 520.506,Z 360.145,A -85,B 0,C 180,E1 25241.351,E2 25241.351} C_VEL
LIN {X 0,Y 520.57,Z 360.143,A -85,B 0,C 180,E1 25238.051,E2 25238.051} C_VEL
LIN {X 0,Y 520.519,Z 360.145,A -85,B 0,C 180,E1 25234.703,E2 25234.703} C_VEL
LIN {X 0,Y 520.508,Z 360.144,A -85,B 0,C 180,E1 25231.234,E2 25231.234} C_VEL
LIN {X 0,Y 520.576,Z 360.143,A -85,B 0,C 180,E1 25227.934,E2 25227.934} C_VEL
LIN {X 0,Y 520.513,Z 360.135,A -85,B 0,C 180,E1 25224.628,E2 25224.628} C_VEL
LIN {X 0,Y 520.513,Z 360.144,A -85,B 0,C 180,E1 25221.163,E2 25221.163} C_VEL
LIN {X 0,Y 520.571,Z 360.125,A -85,B 0,C 180,E1 25217.891,E2 25217.891} C_VEL
LIN {X 0,Y 520.508,Z 360.141,A -85,B 0,C 180,E1 25214.569,E2 25214.569} C_VEL
LIN {X 0,Y 520.516,Z 360.134,A -85,B 0,C 180,E1 25211.069,E2 25211.069} C_VEL
LIN {X 0,Y 520.58,Z 360.13,A -85,B 0,C 180,E1 25207.679,E2 25207.679} C_VEL
LIN {X 0,Y 520.512,Z 360.142,A -85,B 0,C 180,E1 25204.402,E2 25204.402} C_VEL
LIN {X 0,Y 520.513,Z 360.13,A -85,B 0,C 180,E1 25200.876,E2 25200.876} C_VEL
LIN {X 0,Y 520.561,Z 360.143,A -85,B 0,C 180,E1 25197.684,E2 25197.684} C_VEL
LIN {X 0,Y 520.508,Z 360.13,A -85,B 0,C 180,E1 25194.373,E2 25194.373} C_VEL
LIN {X 0,Y 520.543,Z 360.142,A -85,B 0,C 180,E1 25191.045,E2 25191.045} C_VEL
LIN {X 0,Y 520.533,Z 360.142,A -85,B 0,C 180,E1 25187.798,E2 25187.798} C_VEL
LIN {X 0,Y 520.509,Z 360.136,A -85,B 0,C 180,E1 25184.396,E2 25184.396} C_VEL
LIN {X 0,Y 520.563,Z 360.137,A -85,B 0,C 180,E1 25181.055,E2 25181.055} C_VEL
LIN {X 0,Y 520.522,Z 360.129,A -85,B 0,C 180,E1 25177.761,E2 25177.761} C_VEL
LIN {X 0,Y 520.516,Z 360.141,A -85,B 0,C 180,E1 25174.389,E2 25174.389} C_VEL
LIN {X 0,Y 520.577,Z 360.129,A -85,B 0,C 180,E1 25171.049,E2 25171.049} C_VEL
LIN {X 0,Y 520.514,Z 360.142,A -85,B 0,C 180,E1 25167.85,E2 25167.85} C_VEL
LIN {X 0,Y 520.523,Z 360.144,A -85,B 0,C 180,E1 25164.341,E2 25164.341} C_VEL
LIN {X 0,Y 520.567,Z 360.138,A -85,B 0,C 180,E1 25161.065,E2 25161.065} C_VEL
LIN {X 0,Y 520.513,Z 360.141,A -85,B 0,C 180,E1 25157.751,E2 25157.751} C_VEL
LIN {X 0,Y 520.538,Z 360.146,A -85,B 0,C 180,E1 25154.359,E2 25154.359} C_VEL
LIN {X 0,Y 520.546,Z 360.113,A -85,B 0,C 180,E1 25151.063,E2 25151.063} C_VEL
LIN {X 0,Y 520.511,Z 360.128,A -85,B 0,C 180,E1 25147.789,E2 25147.789} C_VEL
LIN {X 0,Y 520.558,Z 360.422,A -85,B 0,C 180,E1 25147.438,E2 25147.438} C_VEL
LIN {X 0,Y 526.109,Z 379.606,A -85,B 0,C 180,E1 25144.362,E2 25144.362} C_VEL
LIN {X 0,Y 525.724,Z 394.479,A -85,B 0,C 180,E1 25142.442,E2 25142.442} C_VEL
LIN {X 0,Y 531.114,Z 414.653,A -85,B 0,C 180,E1 25141.755,E2 25141.755} C_VEL
LIN {X 0,Y 528.862,Z 646.229,A -85,B 0,C 180,E1 25138.338,E2 25138.338} C_VEL
LIN {X 0,Y 528.475,Z 664.061,A -85,B 0,C 180,E1 25137.974,E2 25137.974} C_VEL
LIN {X 0,Y 527.944,Z 681.558,A -85,B 0,C 180,E1 25137.472,E2 25137.472} C_VEL
LIN {X 0,Y 527.144,Z 702.695,A -85,B 0,C 180,E1 25136.652,E2 25136.652} C_VEL
LIN {X 0,Y 526.384,Z 719.042,A -85,B 0,C 180,E1 25135.844,E2 25135.844} C_VEL
LIN {X 0,Y 525.549,Z 735.614,A -85,B 0,C 180,E1 25134.862,E2 25134.862} C_VEL
LIN {X 0,Y 524.513,Z 754.903,A -85,B 0,C 180,E1 25133.478,E2 25133.478} C_VEL
LIN {X 0,Y 523.662,Z 770.141,A -85,B 0,C 180,E1 25132.172,E2 25132.172} C_VEL
LIN {X 0,Y 522.803,Z 785.906,A -85,B 0,C 180,E1 25130.603,E2 25130.603} C_VEL
LIN {X 0,Y 521.999,Z 800.49,A -85,B 0,C 180,E1 25128.872,E2 25128.872} C_VEL
LIN {X 0,Y 521.381,Z 812.81,A -85,B 0,C 180,E1 25127.177,E2 25127.177} C_VEL
LIN {X 0,Y 520.806,Z 826.013,A -85,B 0,C 180,E1 25125.021,E2 25125.021} C_VEL
LIN {X 0,Y 520.434,Z 835.918,A -85,B 0,C 180,E1 25123.078,E2 25123.078} C_VEL
LIN {X 0,Y 520.164,Z 845.434,A -85,B 0,C 180,E1 25120.81,E2 25120.81} C_VEL
LIN {X 0,Y 520.026,Z 852.314,A -85,B 0,C 180,E1 25118.736,E2 25118.736} C_VEL
LIN {X 0,Y 519.947,Z 857.768,A -85,B 0,C 180,E1 25116.625,E2 25116.625} C_VEL
LIN {X 0,Y 519.911,Z 861.928,A -85,B 0,C 180,E1 25114.301,E2 25114.301} C_VEL
LIN {X 0,Y 519.91,Z 864.245,A -85,B 0,C 180,E1 25112.094,E2 25112.094} C_VEL
LIN {X 0,Y 519.902,Z 864.94,A -85,B 0,C 180,E1 25109.669,E2 25109.669} C_VEL
LIN {X 0,Y 519.902,Z 863.983,A -85,B 0,C 180,E1 25107.575,E2 25107.575} C_VEL
LIN {X 0,Y 519.912,Z 861.624,A -85,B 0,C 180,E1 25105.478,E2 25105.478} C_VEL
LIN {X 0,Y 519.959,Z 857.26,A -85,B 0,C 180,E1 25103.153,E2 25103.153} C_VEL
LIN {X 0,Y 520.035,Z 851.654,A -85,B 0,C 180,E1 25101.041,E2 25101.041} C_VEL
LIN {X 0,Y 520.2,Z 844.007,A -85,B 0,C 180,E1 25098.807,E2 25098.807} C_VEL
LIN {X 0,Y 520.457,Z 835.266,A -85,B 0,C 180,E1 25096.785,E2 25096.785} C_VEL
LIN {X 0,Y 520.861,Z 824.777,A -85,B 0,C 180,E1 25094.753,E2 25094.753} C_VEL
LIN {X 0,Y 521.415,Z 812.023,A -85,B 0,C 180,E1 25092.709,E2 25092.709} C_VEL
LIN {X 0,Y 522.05,Z 799.493,A -85,B 0,C 180,E1 25090.999,E2 25090.999} C_VEL
LIN {X 0,Y 522.902,Z 783.7,A -85,B 0,C 180,E1 25089.167,E2 25089.167} C_VEL
LIN {X 0,Y 523.723,Z 769.083,A -85,B 0,C 180,E1 25087.731,E2 25087.731} C_VEL
LIN {X 0,Y 524.663,Z 752.584,A -85,B 0,C 180,E1 25086.335,E2 25086.335} C_VEL
LIN {X 0,Y 525.605,Z 734.36,A -85,B 0,C 180,E1 25085.058,E2 25085.058} C_VEL
LIN {X 0,Y 526.438,Z 717.982,A -85,B 0,C 180,E1 25084.099,E2 25084.099} C_VEL
LIN {X 0,Y 527.316,Z 698.882,A -85,B 0,C 180,E1 25083.175,E2 25083.175} C_VEL
LIN {X 0,Y 528.005,Z 679.615,A -85,B 0,C 180,E1 25082.466,E2 25082.466} C_VEL
LIN {X 0,Y 528.508,Z 662.583,A -85,B 0,C 180,E1 25081.989,E2 25081.989} C_VEL
LIN {X 0,Y 528.949,Z 641.716,A -85,B 0,C 180,E1 25081.586,E2 25081.586} C_VEL
LIN {X 0,Y 531.104,Z 413.917,A -85,B 0,C 180,E1 25078.233,E2 25078.233} C_VEL
LIN {X 0,Y 525.666,Z 393.926,A -85,B 0,C 180,E1 25077.519,E2 25077.519} C_VEL
LIN {X 0,Y 526.107,Z 379.606,A -85,B 0,C 180,E1 25075.638,E2 25075.638} C_VEL
LIN {X 0,Y 520.534,Z 360.275,A -85,B 0,C 180,E1 25072.532,E2 25072.532} C_VEL
LIN {X 0,Y 520.579,Z 360.109,A -85,B 0,C 180,E1 25069.231,E2 25069.231} C_VEL
LIN {X 0,Y 520.518,Z 360.147,A -85,B 0,C 180,E1 25065.926,E2 25065.926} C_VEL
LIN {X 0,Y 520.517,Z 360.141,A -85,B 0,C 180,E1 25062.397,E2 25062.397} C_VEL
LIN {X 0,Y 520.584,Z 360.138,A -85,B 0,C 180,E1 25059.051,E2 25059.051} C_VEL
LIN {X 0,Y 520.519,Z 360.144,A -85,B 0,C 180,E1 25055.732,E2 25055.732} C_VEL
LIN {X 0,Y 520.518,Z 360.142,A -85,B 0,C 180,E1 25052.28,E2 25052.28} C_VEL
LIN {X 0,Y 520.577,Z 360.129,A -85,B 0,C 180,E1 25048.951,E2 25048.951} C_VEL
LIN {X 0,Y 520.516,Z 360.141,A -85,B 0,C 180,E1 25045.611,E2 25045.611} C_VEL
LIN {X 0,Y 520.516,Z 360.129,A -85,B 0,C 180,E1 25042.12,E2 25042.12} C_VEL
LIN {X 0,Y 520.577,Z 360.139,A -85,B 0,C 180,E1 25038.762,E2 25038.762} C_VEL
LIN {X 0,Y 520.512,Z 360.136,A -85,B 0,C 180,E1 25035.49,E2 25035.49} C_VEL
LIN {X 0,Y 520.517,Z 360.141,A -85,B 0,C 180,E1 25031.977,E2 25031.977} C_VEL
LIN {X 0,Y 520.577,Z 360.135,A -85,B 0,C 180,E1 25028.62,E2 25028.62} C_VEL
LIN {X 0,Y 520.508,Z 360.13,A -85,B 0,C 180,E1 25025.405,E2 25025.405} C_VEL
LIN {X 0,Y 520.528,Z 360.143,A -85,B 0,C 180,E1 25021.986,E2 25021.986} C_VEL
LIN {X 0,Y 520.538,Z 360.126,A -85,B 0,C 180,E1 25018.794,E2 25018.794} C_VEL
LIN {X 0,Y 520.509,Z 360.142,A -85,B 0,C 180,E1 25015.488,E2 25015.488} C_VEL
LIN {X 0,Y 520.563,Z 360.129,A -85,B 0,C 180,E1 25012.167,E2 25012.167} C_VEL
LIN {X 0,Y 520.523,Z 360.134,A -85,B 0,C 180,E1 25008.819,E2 25008.819} C_VEL
LIN {X 0,Y 520.508,Z 360.141,A -85,B 0,C 180,E1 25005.431,E2 25005.431} C_VEL
LIN {X 0,Y 520.571,Z 360.125,A -85,B 0,C 180,E1 25002.109,E2 25002.109} C_VEL
LIN {X 0,Y 520.513,Z 360.144,A -85,B 0,C 180,E1 24998.837,E2 24998.837} C_VEL
LIN {X 0,Y 520.511,Z 360.135,A -85,B 0,C 180,E1 24995.308,E2 24995.308} C_VEL
LIN {X 0,Y 520.572,Z 360.144,A -85,B 0,C 180,E1 24991.936,E2 24991.936} C_VEL
LIN {X 0,Y 520.509,Z 360.144,A -85,B 0,C 180,E1 24988.736,E2 24988.736} C_VEL
LIN {X 0,Y 520.514,Z 360.145,A -85,B 0,C 180,E1 24985.223,E2 24985.223} C_VEL
LIN {X 0,Y 520.571,Z 360.143,A -85,B 0,C 180,E1 24981.945,E2 24981.945} C_VEL
LIN {X 0,Y 520.506,Z 360.145,A -85,B 0,C 180,E1 24978.649,E2 24978.649} C_VEL
LIN {X 0,Y 520.565,Z 360.144,A -85,B 0,C 180,E1 24977.898,E2 24977.898} C_VEL
LIN {X 0,Y 519.732,Z 360.249,A -85,B 0,C 180,E1 24977.11,E2 24977.11} C_VEL
LIN {X 0,Y 515.463,Z 360.779,A -85,B 0,C 180,E1 24975.634,E2 24975.634} C_VEL
LIN {X 0,Y 512.838,Z 361.101,A -85,B 0,C 180,E1 24974.483,E2 24974.483} C_VEL
LIN {X 0,Y 512.603,Z 361.134,A -85,B 0,C 180,E1 24974.047,E2 24974.047} C_VEL
LIN {X 0,Y 512.565,Z 361.133,A -85,B 0,C 180,E1 24970.656,E2 24970.656} C_VEL
LIN {X 0,Y 512.601,Z 361.134,A -85,B 0,C 180,E1 24967.28,E2 24967.28} C_VEL
LIN {X 0,Y 512.589,Z 361.134,A -85,B 0,C 180,E1 24964.018,E2 24964.018} C_VEL
LIN {X 0,Y 512.565,Z 361.134,A -85,B 0,C 180,E1 24960.605,E2 24960.605} C_VEL
LIN {X 0,Y 512.62,Z 361.132,A -85,B 0,C 180,E1 24957.281,E2 24957.281} C_VEL
LIN {X 0,Y 512.581,Z 361.135,A -85,B 0,C 180,E1 24953.936,E2 24953.936} C_VEL
LIN {X 0,Y 512.568,Z 361.133,A -85,B 0,C 180,E1 24950.555,E2 24950.555} C_VEL
LIN {X 0,Y 512.629,Z 361.132,A -85,B 0,C 180,E1 24947.245,E2 24947.245} C_VEL
LIN {X 0,Y 512.568,Z 361.135,A -85,B 0,C 180,E1 24943.997,E2 24943.997} C_VEL
LIN {X 0,Y 512.57,Z 361.135,A -85,B 0,C 180,E1 24940.452,E2 24940.452} C_VEL
LIN {X 0,Y 512.635,Z 361.131,A -85,B 0,C 180,E1 24937.058,E2 24937.058} C_VEL
LIN {X 0,Y 512.573,Z 361.134,A -85,B 0,C 180,E1 24933.691,E2 24933.691} C_VEL
LIN {X 0,Y 512.566,Z 361.136,A -85,B 0,C 180,E1 24930.224,E2 24930.224} C_VEL
LIN {X 0,Y 512.622,Z 361.135,A -85,B 0,C 180,E1 24926.869,E2 24926.869} C_VEL
LIN {X 0,Y 512.576,Z 361.135,A -85,B 0,C 180,E1 24923.504,E2 24923.504} C_VEL
LIN {X 0,Y 512.565,Z 361.135,A -85,B 0,C 180,E1 24920.002,E2 24920.002} C_VEL
LIN {X 0,Y 512.627,Z 361.132,A -85,B 0,C 180,E1 24916.686,E2 24916.686} C_VEL
LIN {X 0,Y 512.571,Z 361.135,A -85,B 0,C 180,E1 24913.454,E2 24913.454} C_VEL
LIN {X 0,Y 512.569,Z 361.133,A -85,B 0,C 180,E1 24909.921,E2 24909.921} C_VEL
LIN {X 0,Y 512.633,Z 361.132,A -85,B 0,C 180,E1 24906.676,E2 24906.676} C_VEL
LIN {X 0,Y 512.571,Z 361.135,A -85,B 0,C 180,E1 24903.286,E2 24903.286} C_VEL
LIN {X 0,Y 512.572,Z 361.133,A -85,B 0,C 180,E1 24899.769,E2 24899.769} C_VEL
LIN {X 0,Y 512.631,Z 361.132,A -85,B 0,C 180,E1 24896.499,E2 24896.499} C_VEL
LIN {X 0,Y 512.568,Z 361.135,A -85,B 0,C 180,E1 24893.213,E2 24893.213} C_VEL
LIN {X 0,Y 512.574,Z 361.133,A -85,B 0,C 180,E1 24889.691,E2 24889.691} C_VEL
LIN {X 0,Y 512.618,Z 361.134,A -85,B 0,C 180,E1 24886.488,E2 24886.488} C_VEL
LIN {X 0,Y 512.567,Z 361.134,A -85,B 0,C 180,E1 24883.153,E2 24883.153} C_VEL
LIN {X 0,Y 512.595,Z 361.133,A -85,B 0,C 180,E1 24879.766,E2 24879.766} C_VEL
LIN {X 0,Y 512.595,Z 361.133,A -85,B 0,C 180,E1 24876.523,E2 24876.523} C_VEL
LIN {X 0,Y 512.57,Z 361.134,A -85,B 0,C 180,E1 24873.195,E2 24873.195} C_VEL
LIN {X 0,Y 512.619,Z 361.133,A -85,B 0,C 180,E1 24869.818,E2 24869.818} C_VEL
LIN {X 0,Y 512.584,Z 361.134,A -85,B 0,C 180,E1 24866.524,E2 24866.524} C_VEL
LIN {X 0,Y 512.57,Z 361.123,A -85,B 0,C 180,E1 24863.077,E2 24863.077} C_VEL
LIN {X 0,Y 512.633,Z 361.128,A -85,B 0,C 180,E1 24859.832,E2 24859.832} C_VEL
LIN {X 0,Y 512.571,Z 361.113,A -85,B 0,C 180,E1 24856.54,E2 24856.54} C_VEL
LIN {X 0,Y 512.572,Z 361.133,A -85,B 0,C 180,E1 24852.957,E2 24852.957} C_VEL
LIN {X 0,Y 512.629,Z 361.108,A -85,B 0,C 180,E1 24849.651,E2 24849.651} C_VEL
LIN {X 0,Y 512.574,Z 361.131,A -85,B 0,C 180,E1 24846.378,E2 24846.378} C_VEL
LIN {X 0,Y 512.575,Z 361.119,A -85,B 0,C 180,E1 24842.902,E2 24842.902} C_VEL
LIN {X 0,Y 512.641,Z 361.119,A -85,B 0,C 180,E1 24839.548,E2 24839.548} C_VEL
LIN {X 0,Y 512.577,Z 361.131,A -85,B 0,C 180,E1 24836.193,E2 24836.193} C_VEL
LIN {X 0,Y 512.576,Z 361.12,A -85,B 0,C 180,E1 24832.711,E2 24832.711} C_VEL
LIN {X 0,Y 512.632,Z 361.133,A -85,B 0,C 180,E1 24829.418,E2 24829.418} C_VEL
LIN {X 0,Y 512.571,Z 361.115,A -85,B 0,C 180,E1 24826.113,E2 24826.113} C_VEL
LIN {X 0,Y 512.581,Z 361.133,A -85,B 0,C 180,E1 24822.632,E2 24822.632} C_VEL
LIN {X 0,Y 512.63,Z 361.113,A -85,B 0,C 180,E1 24819.324,E2 24819.324} C_VEL
LIN {X 0,Y 512.572,Z 361.132,A -85,B 0,C 180,E1 24816.059,E2 24816.059} C_VEL
LIN {X 0,Y 512.602,Z 361.113,A -85,B 0,C 180,E1 24812.714,E2 24812.714} C_VEL
LIN {X 0,Y 512.593,Z 361.132,A -85,B 0,C 180,E1 24809.522,E2 24809.522} C_VEL
LIN {X 0,Y 512.573,Z 361.126,A -85,B 0,C 180,E1 24806.087,E2 24806.087} C_VEL
LIN {X 0,Y 512.621,Z 361.121,A -85,B 0,C 180,E1 24802.728,E2 24802.728} C_VEL
LIN {X 0,Y 512.585,Z 361.134,A -85,B 0,C 180,E1 24799.489,E2 24799.489} C_VEL
LIN {X 0,Y 512.576,Z 361.132,A -85,B 0,C 180,E1 24796.015,E2 24796.015} C_VEL
LIN {X 0,Y 512.631,Z 361.12,A -85,B 0,C 180,E1 24792.663,E2 24792.663} C_VEL
LIN {X 0,Y 512.584,Z 361.124,A -85,B 0,C 180,E1 24789.341,E2 24789.341} C_VEL
LIN {X 0,Y 512.619,Z 361.413,A -85,B 0,C 180,E1 24787.934,E2 24787.934} C_VEL
LIN {X 0,Y 517.769,Z 378.994,A -85,B 0,C 180,E1 24785.035,E2 24785.035} C_VEL
LIN {X 0,Y 518.732,Z 383.694,A -85,B 0,C 180,E1 24784.318,E2 24784.318} C_VEL
LIN {X 0,Y 518.347,Z 394.161,A -85,B 0,C 180,E1 24782.964,E2 24782.964} C_VEL
LIN {X 0,Y 524.28,Z 416.449,A -85,B 0,C 180,E1 24782.187,E2 24782.187} C_VEL
LIN {X 0,Y 521.798,Z 646.608,A -85,B 0,C 180,E1 24778.745,E2 24778.745} C_VEL
LIN {X 0,Y 521.372,Z 664.255,A -85,B 0,C 180,E1 24778.379,E2 24778.379} C_VEL
LIN {X 0,Y 520.776,Z 682.303,A -85,B 0,C 180,E1 24777.852,E2 24777.852} C_VEL
LIN {X 0,Y 519.901,Z 703.163,A -85,B 0,C 180,E1 24777.025,E2 24777.025} C_VEL
LIN {X 0,Y 519.11,Z 718.97,A -85,B 0,C 180,E1 24776.236,E2 24776.236} C_VEL
LIN {X 0,Y 518.22,Z 734.946,A -85,B 0,C 180,E1 24775.282,E2 24775.282} C_VEL
LIN {X 0,Y 517.149,Z 753.476,A -85,B 0,C 180,E1 24773.954,E2 24773.954} C_VEL
LIN {X 0,Y 516.174,Z 769.002,A -85,B 0,C 180,E1 24772.619,E2 24772.619} C_VEL
LIN {X 0,Y 515.283,Z 783.293,A -85,B 0,C 180,E1 24771.199,E2 24771.199} C_VEL
LIN {X 0,Y 514.369,Z 798.6,A -85,B 0,C 180,E1 24769.414,E2 24769.414} C_VEL
LIN {X 0,Y 513.652,Z 811.232,A -85,B 0,C 180,E1 24767.677,E2 24767.677} C_VEL
LIN {X 0,Y 513.046,Z 823.501,A -85,B 0,C 180,E1 24765.717,E2 24765.717} C_VEL
LIN {X 0,Y 512.581,Z 834.187,A -85,B 0,C 180,E1 24763.652,E2 24763.652} C_VEL
LIN {X 0,Y 512.282,Z 842.62,A -85,B 0,C 180,E1 24761.711,E2 24761.711} C_VEL
LIN {X 0,Y 512.071,Z 850.989,A -85,B 0,C 180,E1 24759.326,E2 24759.326} C_VEL
LIN {X 0,Y 511.973,Z 856.722,A -85,B 0,C 180,E1 24757.18,E2 24757.18} C_VEL
LIN {X 0,Y 511.928,Z 861.151,A -85,B 0,C 180,E1 24754.93,E2 24754.93} C_VEL
LIN {X 0,Y 511.908,Z 863.804,A -85,B 0,C 180,E1 24752.687,E2 24752.687} C_VEL
LIN {X 0,Y 511.901,Z 864.888,A -85,B 0,C 180,E1 24750.56,E2 24750.56} C_VEL
LIN {X 0,Y 511.908,Z 864.472,A -85,B 0,C 180,E1 24748.209,E2 24748.209} C_VEL
LIN {X 0,Y 511.916,Z 862.361,A -85,B 0,C 180,E1 24745.968,E2 24745.968} C_VEL
LIN {X 0,Y 511.942,Z 859.116,A -85,B 0,C 180,E1 24743.946,E2 24743.946} C_VEL
LIN {X 0,Y 512.016,Z 853.629,A -85,B 0,C 180,E1 24741.578,E2 24741.578} C_VEL
LIN {X 0,Y 512.163,Z 846.854,A -85,B 0,C 180,E1 24739.426,E2 24739.426} C_VEL
LIN {X 0,Y 512.428,Z 838.428,A -85,B 0,C 180,E1 24737.263,E2 24737.263} C_VEL
LIN {X 0,Y 512.81,Z 828.462,A -85,B 0,C 180,E1 24735.202,E2 24735.202} C_VEL
LIN {X 0,Y 513.308,Z 817.959,A -85,B 0,C 180,E1 24733.362,E2 24733.362} C_VEL
LIN {X 0,Y 514.07,Z 803.909,A -85,B 0,C 180,E1 24731.282,E2 24731.282} C_VEL
LIN {X 0,Y 514.847,Z 790.417,A -85,B 0,C 180,E1 24729.599,E2 24729.599} C_VEL
LIN {X 0,Y 515.836,Z 774.702,A -85,B 0,C 180,E1 24727.912,E2 24727.912} C_VEL
LIN {X 0,Y 516.824,Z 758.506,A -85,B 0,C 180,E1 24726.46,E2 24726.46} C_VEL
LIN {X 0,Y 517.748,Z 743.275,A -85,B 0,C 180,E1 24725.286,E2 24725.286} C_VEL
LIN {X 0,Y 518.839,Z 724.325,A -85,B 0,C 180,E1 24724.059,E2 24724.059} C_VEL
LIN {X 0,Y 519.724,Z 706.706,A -85,B 0,C 180,E1 24723.14,E2 24723.14} C_VEL
LIN {X 0,Y 520.466,Z 689.846,A -85,B 0,C 180,E1 24722.421,E2 24722.421} C_VEL
LIN {X 0,Y 521.257,Z 669.005,A -85,B 0,C 180,E1 24721.74,E2 24721.74} C_VEL
LIN {X 0,Y 521.73,Z 650.102,A -85,B 0,C 180,E1 24721.317,E2 24721.317} C_VEL
LIN {X 0,Y 524.192,Z 424.803,A -85,B 0,C 180,E1 24717.94,E2 24717.94} C_VEL
LIN {X 0,Y 524.081,Z 414.99,A -85,B 0,C 180,E1 24717.777,E2 24717.777} C_VEL
LIN {X 0,Y 518.293,Z 393.711,A -85,B 0,C 180,E1 24717.005,E2 24717.005} C_VEL
LIN {X 0,Y 518.643,Z 382.231,A -85,B 0,C 180,E1 24715.475,E2 24715.475} C_VEL
LIN {X 0,Y 513.233,Z 363.475,A -85,B 0,C 180,E1 24712.428,E2 24712.428} C_VEL
LIN {X 0,Y 512.589,Z 361.191,A -85,B 0,C 180,E1 24712.006,E2 24712.006} C_VEL
LIN {X 0,Y 512.573,Z 361.108,A -85,B 0,C 180,E1 24708.455,E2 24708.455} C_VEL
LIN {X 0,Y 512.632,Z 361.124,A -85,B 0,C 180,E1 24705.087,E2 24705.087} C_VEL
LIN {X 0,Y 512.58,Z 361.128,A -85,B 0,C 180,E1 24701.83,E2 24701.83} C_VEL
LIN {X 0,Y 512.578,Z 361.125,A -85,B 0,C 180,E1 24698.341,E2 24698.341} C_VEL
LIN {X 0,Y 512.637,Z 361.129,A -85,B 0,C 180,E1 24694.992,E2 24694.992} C_VEL
LIN {X 0,Y 512.581,Z 361.131,A -85,B 0,C 180,E1 24691.653,E2 24691.653} C_VEL
LIN {X 0,Y 512.575,Z 361.114,A -85,B 0,C 180,E1 24688.156,E2 24688.156} C_VEL
LIN {X 0,Y 512.634,Z 361.133,A -85,B 0,C 180,E1 24684.797,E2 24684.797} C_VEL
LIN {X 0,Y 512.578,Z 361.116,A -85,B 0,C 180,E1 24681.498,E2 24681.498} C_VEL
LIN {X 0,Y 512.573,Z 361.133,A -85,B 0,C 180,E1 24677.955,E2 24677.955} C_VEL
LIN {X 0,Y 512.629,Z 361.109,A -85,B 0,C 180,E1 24674.577,E2 24674.577} C_VEL
LIN {X 0,Y 512.583,Z 361.13,A -85,B 0,C 180,E1 24671.253,E2 24671.253} C_VEL
LIN {X 0,Y 512.574,Z 361.12,A -85,B 0,C 180,E1 24667.852,E2 24667.852} C_VEL
LIN {X 0,Y 512.632,Z 361.118,A -85,B 0,C 180,E1 24664.591,E2 24664.591} C_VEL
LIN {X 0,Y 512.575,Z 361.131,A -85,B 0,C 180,E1 24661.234,E2 24661.234} C_VEL
LIN {X 0,Y 512.572,Z 361.119,A -85,B 0,C 180,E1 24657.657,E2 24657.657} C_VEL
LIN {X 0,Y 512.634,Z 361.132,A -85,B 0,C 180,E1 24654.297,E2 24654.297} C_VEL
LIN {X 0,Y 512.574,Z 361.116,A -85,B 0,C 180,E1 24651.028,E2 24651.028} C_VEL
LIN {X 0,Y 512.573,Z 361.133,A -85,B 0,C 180,E1 24647.501,E2 24647.501} C_VEL
LIN {X 0,Y 512.634,Z 361.114,A -85,B 0,C 180,E1 24644.16,E2 24644.16} C_VEL
LIN {X 0,Y 512.581,Z 361.127,A -85,B 0,C 180,E1 24640.748,E2 24640.748} C_VEL
LIN {X 0,Y 512.57,Z 361.124,A -85,B 0,C 180,E1 24637.287,E2 24637.287} C_VEL
LIN {X 0,Y 512.629,Z 361.126,A -85,B 0,C 180,E1 24633.977,E2 24633.977} C_VEL
LIN {X 0,Y 512.575,Z 361.133,A -85,B 0,C 180,E1 24630.682,E2 24630.682} C_VEL
LIN {X 0,Y 512.572,Z 361.134,A -85,B 0,C 180,E1 24627.169,E2 24627.169} C_VEL
LIN {X 0,Y 512.628,Z 361.133,A -85,B 0,C 180,E1 24623.782,E2 24623.782} C_VEL
LIN {X 0,Y 512.573,Z 361.133,A -85,B 0,C 180,E1 24620.522,E2 24620.522} C_VEL
LIN {X 0,Y 512.571,Z 361.134,A -85,B 0,C 180,E1 24617.011,E2 24617.011} C_VEL
LIN {X 0,Y 512.603,Z 361.134,A -85,B 0,C 180,E1 24614.047,E2 24614.047} C_VEL
LIN {X 0,Y 511.788,Z 361.24,A -85,B 0,C 180,E1 24613.247,E2 24613.247} C_VEL
LIN {X 0,Y 507.718,Z 361.744,A -85,B 0,C 180,E1 24611.807,E2 24611.807} C_VEL
LIN {X 0,Y 504.972,Z 362.08,A -85,B 0,C 180,E1 24610.641,E2 24610.641} C_VEL
LIN {X 0,Y 504.648,Z 362.122,A -85,B 0,C 180,E1 24610.135,E2 24610.135} C_VEL
LIN {X 0,Y 504.629,Z 362.123,A -85,B 0,C 180,E1 24606.752,E2 24606.752} C_VEL
LIN {X 0,Y 504.687,Z 362.121,A -85,B 0,C 180,E1 24603.418,E2 24603.418} C_VEL
LIN {X 0,Y 504.642,Z 362.123,A -85,B 0,C 180,E1 24600.039,E2 24600.039} C_VEL
LIN {X 0,Y 504.629,Z 362.124,A -85,B 0,C 180,E1 24596.601,E2 24596.601} C_VEL
LIN {X 0,Y 504.682,Z 362.123,A -85,B 0,C 180,E1 24593.204,E2 24593.204} C_VEL
LIN {X 0,Y 504.638,Z 362.122,A -85,B 0,C 180,E1 24589.924,E2 24589.924} C_VEL
LIN {X 0,Y 504.629,Z 362.125,A -85,B 0,C 180,E1 24586.459,E2 24586.459} C_VEL
LIN {X 0,Y 504.691,Z 362.122,A -85,B 0,C 180,E1 24583.169,E2 24583.169} C_VEL
LIN {X 0,Y 504.634,Z 362.124,A -85,B 0,C 180,E1 24579.811,E2 24579.811} C_VEL
LIN {X 0,Y 504.63,Z 362.124,A -85,B 0,C 180,E1 24576.37,E2 24576.37} C_VEL
LIN {X 0,Y 504.683,Z 362.122,A -85,B 0,C 180,E1 24572.953,E2 24572.953} C_VEL
LIN {X 0,Y 504.632,Z 362.125,A -85,B 0,C 180,E1 24569.659,E2 24569.659} C_VEL
LIN {X 0,Y 504.627,Z 362.123,A -85,B 0,C 180,E1 24566.137,E2 24566.137} C_VEL
LIN {X 0,Y 504.694,Z 362.12,A -85,B 0,C 180,E1 24562.83,E2 24562.83} C_VEL
LIN {X 0,Y 504.634,Z 362.124,A -85,B 0,C 180,E1 24559.497,E2 24559.497} C_VEL
LIN {X 0,Y 504.63,Z 362.124,A -85,B 0,C 180,E1 24556.012,E2 24556.012} C_VEL
LIN {X 0,Y 504.69,Z 362.121,A -85,B 0,C 180,E1 24552.698,E2 24552.698} C_VEL
LIN {X 0,Y 504.633,Z 362.122,A -85,B 0,C 180,E1 24549.349,E2 24549.349} C_VEL
LIN {X 0,Y 504.63,Z 362.124,A -85,B 0,C 180,E1 24545.787,E2 24545.787} C_VEL
LIN {X 0,Y 504.682,Z 362.123,A -85,B 0,C 180,E1 24542.382,E2 24542.382} C_VEL
LIN {X 0,Y 504.641,Z 362.123,A -85,B 0,C 180,E1 24539.067,E2 24539.067} C_VEL
LIN {X 0,Y 504.63,Z 362.124,A -85,B 0,C 180,E1 24535.62,E2 24535.62} C_VEL
LIN {X 0,Y 504.681,Z 362.122,A -85,B 0,C 180,E1 24532.218,E2 24532.218} C_VEL
LIN {X 0,Y 504.645,Z 362.122,A -85,B 0,C 180,E1 24528.87,E2 24528.87} C_VEL
LIN {X 0,Y 504.63,Z 362.123,A -85,B 0,C 180,E1 24525.462,E2 24525.462} C_VEL
LIN {X 0,Y 504.695,Z 362.121,A -85,B 0,C 180,E1 24522.18,E2 24522.18} C_VEL
LIN {X 0,Y 504.635,Z 362.122,A -85,B 0,C 180,E1 24518.863,E2 24518.863} C_VEL
LIN {X 0,Y 504.631,Z 362.123,A -85,B 0,C 180,E1 24515.284,E2 24515.284} C_VEL
LIN {X 0,Y 504.688,Z 362.122,A -85,B 0,C 180,E1 24511.927,E2 24511.927} C_VEL
LIN {X 0,Y 504.641,Z 362.122,A -85,B 0,C 180,E1 24508.634,E2 24508.634} C_VEL
LIN {X 0,Y 504.63,Z 362.111,A -85,B 0,C 180,E1 24505.115,E2 24505.115} C_VEL
LIN {X 0,Y 504.681,Z 362.12,A -85,B 0,C 180,E1 24501.699,E2 24501.699} C_VEL
LIN {X 0,Y 504.648,Z 362.114,A -85,B 0,C 180,E1 24498.356,E2 24498.356} C_VEL
LIN {X 0,Y 504.629,Z 362.118,A -85,B 0,C 180,E1 24494.92,E2 24494.92} C_VEL
LIN {X 0,Y 504.689,Z 362.111,A -85,B 0,C 180,E1 24491.652,E2 24491.652} C_VEL
LIN {X 0,Y 504.64,Z 362.104,A -85,B 0,C 180,E1 24488.311,E2 24488.311} C_VEL
LIN {X 0,Y 504.633,Z 362.12,A -85,B 0,C 180,E1 24484.768,E2 24484.768} C_VEL
LIN {X 0,Y 504.676,Z 362.097,A -85,B 0,C 180,E1 24481.357,E2 24481.357} C_VEL
LIN {X 0,Y 504.647,Z 362.12,A -85,B 0,C 180,E1 24478.065,E2 24478.065} C_VEL
LIN {X 0,Y 504.633,Z 362.105,A -85,B 0,C 180,E1 24474.652,E2 24474.652} C_VEL
LIN {X 0,Y 504.694,Z 362.112,A -85,B 0,C 180,E1 24471.32,E2 24471.32} C_VEL
LIN {X 0,Y 504.641,Z 362.119,A -85,B 0,C 180,E1 24467.988,E2 24467.988} C_VEL
LIN {X 0,Y 504.634,Z 362.113,A -85,B 0,C 180,E1 24464.481,E2 24464.481} C_VEL
LIN {X 0,Y 504.693,Z 362.115,A -85,B 0,C 180,E1 24461.156,E2 24461.156} C_VEL
LIN {X 0,Y 504.645,Z 362.105,A -85,B 0,C 180,E1 24457.76,E2 24457.76} C_VEL
LIN {X 0,Y 504.635,Z 362.119,A -85,B 0,C 180,E1 24454.28,E2 24454.28} C_VEL
LIN {X 0,Y 504.686,Z 362.109,A -85,B 0,C 180,E1 24450.887,E2 24450.887} C_VEL
LIN {X 0,Y 504.653,Z 362.119,A -85,B 0,C 180,E1 24447.522,E2 24447.522} C_VEL
LIN {X 0,Y 504.635,Z 362.122,A -85,B 0,C 180,E1 24444.089,E2 24444.089} C_VEL
LIN {X 0,Y 504.693,Z 362.12,A -85,B 0,C 180,E1 24440.768,E2 24440.768} C_VEL
LIN {X 0,Y 504.645,Z 362.119,A -85,B 0,C 180,E1 24437.479,E2 24437.479} C_VEL
LIN {X 0,Y 504.639,Z 362.126,A -85,B 0,C 180,E1 24434.007,E2 24434.007} C_VEL
LIN {X 0,Y 504.694,Z 362.082,A -85,B 0,C 180,E1 24430.642,E2 24430.642} C_VEL
LIN {X 0,Y 504.716,Z 362.382,A -85,B 0,C 180,E1 24428.45,E2 24428.45} C_VEL
LIN {X 0,Y 509.821,Z 379.921,A -85,B 0,C 180,E1 24425.485,E2 24425.485} C_VEL
LIN {X 0,Y 511.302,Z 385.825,A -85,B 0,C 180,E1 24424.547,E2 24424.547} C_VEL
LIN {X 0,Y 511.004,Z 393.904,A -85,B 0,C 180,E1 24423.5,E2 24423.5} C_VEL
LIN {X 0,Y 517.476,Z 418.315,A -85,B 0,C 180,E1 24422.628,E2 24422.628} C_VEL
LIN {X 0,Y 514.758,Z 647.09,A -85,B 0,C 180,E1 24419.162,E2 24419.162} C_VEL
LIN {X 0,Y 514.288,Z 664.641,A -85,B 0,C 180,E1 24418.789,E2 24418.789} C_VEL
LIN {X 0,Y 513.583,Z 684.221,A -85,B 0,C 180,E1 24418.202,E2 24418.202} C_VEL
LIN {X 0,Y 512.657,Z 703.609,A -85,B 0,C 180,E1 24417.404,E2 24417.404} C_VEL
LIN {X 0,Y 511.768,Z 719.845,A -85,B 0,C 180,E1 24416.576,E2 24416.576} C_VEL
LIN {X 0,Y 510.779,Z 736.365,A -85,B 0,C 180,E1 24415.57,E2 24415.57} C_VEL
LIN {X 0,Y 509.603,Z 754.855,A -85,B 0,C 180,E1 24414.208,E2 24414.208} C_VEL
LIN {X 0,Y 508.633,Z 769.063,A -85,B 0,C 180,E1 24412.967,E2 24412.967} C_VEL
LIN {X 0,Y 507.68,Z 783.129,A -85,B 0,C 180,E1 24411.549,E2 24411.549} C_VEL
LIN {X 0,Y 506.654,Z 798.608,A -85,B 0,C 180,E1 24409.72,E2 24409.72} C_VEL
LIN {X 0,Y 505.904,Z 810.453,A -85,B 0,C 180,E1 24408.074,E2 24408.074} C_VEL
LIN {X 0,Y 505.283,Z 821.468,A -85,B 0,C 180,E1 24406.314,E2 24406.314} C_VEL
LIN {X 0,Y 504.711,Z 833.108,A -85,B 0,C 180,E1 24404.103,E2 24404.103} C_VEL
LIN {X 0,Y 504.353,Z 841.688,A -85,B 0,C 180,E1 24402.13,E2 24402.13} C_VEL
LIN {X 0,Y 504.119,Z 849.603,A -85,B 0,C 180,E1 24399.936,E2 24399.936} C_VEL
LIN {X 0,Y 503.99,Z 855.916,A -85,B 0,C 180,E1 24397.638,E2 24397.638} C_VEL
LIN {X 0,Y 503.933,Z 860.142,A -85,B 0,C 180,E1 24395.579,E2 24395.579} C_VEL
LIN {X 0,Y 503.913,Z 863.433,A -85,B 0,C 180,E1 24393.185,E2 24393.185} C_VEL
LIN {X 0,Y 503.912,Z 864.797,A -85,B 0,C 180,E1 24390.909,E2 24390.909} C_VEL
LIN {X 0,Y 503.91,Z 864.739,A -85,B 0,C 180,E1 24388.863,E2 24388.863} C_VEL
LIN {X 0,Y 503.912,Z 863.033,A -85,B 0,C 180,E1 24386.432,E2 24386.432} C_VEL
LIN {X 0,Y 503.936,Z 859.936,A -85,B 0,C 180,E1 24384.307,E2 24384.307} C_VEL
LIN {X 0,Y 503.996,Z 855.649,A -85,B 0,C 180,E1 24382.247,E2 24382.247} C_VEL
LIN {X 0,Y 504.135,Z 848.827,A -85,B 0,C 180,E1 24379.833,E2 24379.833} C_VEL
LIN {X 0,Y 504.365,Z 841.331,A -85,B 0,C 180,E1 24377.781,E2 24377.781} C_VEL
LIN {X 0,Y 504.765,Z 832.034,A -85,B 0,C 180,E1 24375.665,E2 24375.665} C_VEL
LIN {X 0,Y 505.319,Z 820.741,A -85,B 0,C 180,E1 24373.564,E2 24373.564} C_VEL
LIN {X 0,Y 505.904,Z 810.44,A -85,B 0,C 180,E1 24371.924,E2 24371.924} C_VEL
LIN {X 0,Y 506.721,Z 797.707,A -85,B 0,C 180,E1 24370.161,E2 24370.161} C_VEL
LIN {X 0,Y 507.739,Z 782.234,A -85,B 0,C 180,E1 24368.357,E2 24368.357} C_VEL
LIN {X 0,Y 508.672,Z 768.435,A -85,B 0,C 180,E1 24366.974,E2 24366.974} C_VEL
LIN {X 0,Y 509.823,Z 752.001,A -85,B 0,C 180,E1 24365.556,E2 24365.556} C_VEL
LIN {X 0,Y 510.883,Z 734.519,A -85,B 0,C 180,E1 24364.311,E2 24364.311} C_VEL
LIN {X 0,Y 511.8,Z 719.293,A -85,B 0,C 180,E1 24363.393,E2 24363.393} C_VEL
LIN {X 0,Y 512.72,Z 702.4,A -85,B 0,C 180,E1 24362.538,E2 24362.538} C_VEL
LIN {X 0,Y 513.696,Z 681.033,A -85,B 0,C 180,E1 24361.694,E2 24361.694} C_VEL
LIN {X 0,Y 514.317,Z 663.528,A -85,B 0,C 180,E1 24361.183,E2 24361.183} C_VEL
LIN {X 0,Y 514.806,Z 645.138,A -85,B 0,C 180,E1 24360.803,E2 24360.803} C_VEL
LIN {X 0,Y 517.471,Z 417.467,A -85,B 0,C 180,E1 24357.358,E2 24357.358} C_VEL
LIN {X 0,Y 510.942,Z 393.382,A -85,B 0,C 180,E1 24356.464,E2 24356.464} C_VEL
LIN {X 0,Y 511.182,Z 384.847,A -85,B 0,C 180,E1 24355.308,E2 24355.308} C_VEL
LIN {X 0,Y 506.106,Z 367.113,A -85,B 0,C 180,E1 24352.379,E2 24352.379} C_VEL
LIN {X 0,Y 504.692,Z 362.178,A -85,B 0,C 180,E1 24351.497,E2 24351.497} C_VEL
LIN {X 0,Y 504.632,Z 362.098,A -85,B 0,C 180,E1 24348.161,E2 24348.161} C_VEL
LIN {X 0,Y 504.655,Z 362.117,A -85,B 0,C 180,E1 24344.699,E2 24344.699} C_VEL
LIN {X 0,Y 504.69,Z 362.111,A -85,B 0,C 180,E1 24341.281,E2 24341.281} C_VEL
LIN {X 0,Y 504.635,Z 362.113,A -85,B 0,C 180,E1 24337.898,E2 24337.898} C_VEL
LIN {X 0,Y 504.643,Z 362.115,A -85,B 0,C 180,E1 24334.383,E2 24334.383} C_VEL
LIN {X 0,Y 504.7,Z 362.121,A -85,B 0,C 180,E1 24330.931,E2 24330.931} C_VEL
LIN {X 0,Y 504.638,Z 362.101,A -85,B 0,C 180,E1 24327.625,E2 24327.625} C_VEL
LIN {X 0,Y 504.637,Z 362.121,A -85,B 0,C 180,E1 24324.093,E2 24324.093} C_VEL
LIN {X 0,Y 504.696,Z 362.099,A -85,B 0,C 180,E1 24320.763,E2 24320.763} C_VEL
LIN {X 0,Y 504.641,Z 362.122,A -85,B 0,C 180,E1 24317.412,E2 24317.412} C_VEL
LIN {X 0,Y 504.632,Z 362.102,A -85,B 0,C 180,E1 24313.871,E2 24313.871} C_VEL
LIN {X 0,Y 504.688,Z 362.122,A -85,B 0,C 180,E1 24310.506,E2 24310.506} C_VEL
LIN {X 0,Y 504.642,Z 362.106,A -85,B 0,C 180,E1 24307.175,E2 24307.175} C_VEL
LIN {X 0,Y 504.632,Z 362.12,A -85,B 0,C 180,E1 24303.64,E2 24303.64} C_VEL
LIN {X 0,Y 504.675,Z 362.107,A -85,B 0,C 180,E1 24300.232,E2 24300.232} C_VEL
LIN {X 0,Y 504.656,Z 362.106,A -85,B 0,C 180,E1 24296.825,E2 24296.825} C_VEL
LIN {X 0,Y 504.629,Z 362.119,A -85,B 0,C 180,E1 24293.406,E2 24293.406} C_VEL
LIN {X 0,Y 504.675,Z 362.099,A -85,B 0,C 180,E1 24290.08,E2 24290.08} C_VEL
LIN {X 0,Y 504.653,Z 362.121,A -85,B 0,C 180,E1 24286.719,E2 24286.719} C_VEL
LIN {X 0,Y 504.628,Z 362.1,A -85,B 0,C 180,E1 24283.31,E2 24283.31} C_VEL
LIN {X 0,Y 504.683,Z 362.122,A -85,B 0,C 180,E1 24279.963,E2 24279.963} C_VEL
LIN {X 0,Y 504.643,Z 362.11,A -85,B 0,C 180,E1 24276.662,E2 24276.662} C_VEL
LIN {X 0,Y 504.631,Z 362.123,A -85,B 0,C 180,E1 24273.152,E2 24273.152} C_VEL
LIN {X 0,Y 504.677,Z 362.123,A -85,B 0,C 180,E1 24269.743,E2 24269.743} C_VEL
LIN {X 0,Y 504.646,Z 362.123,A -85,B 0,C 180,E1 24266.45,E2 24266.45} C_VEL
LIN {X 0,Y 504.63,Z 362.121,A -85,B 0,C 180,E1 24262.972,E2 24262.972} C_VEL
LIN {X 0,Y 504.681,Z 362.121,A -85,B 0,C 180,E1 24259.631,E2 24259.631} C_VEL
LIN {X 0,Y 504.647,Z 362.123,A -85,B 0,C 180,E1 24256.264,E2 24256.264} C_VEL
LIN {X 0,Y 504.629,Z 362.123,A -85,B 0,C 180,E1 24252.812,E2 24252.812} C_VEL
LIN {X 0,Y 504.648,Z 362.122,A -85,B 0,C 180,E1 24250.135,E2 24250.135} C_VEL
LIN {X 0,Y 503.693,Z 362.245,A -85,B 0,C 180,E1 24249.26,E2 24249.26} C_VEL
LIN {X 0,Y 497.212,Z 363.049,A -85,B 0,C 180,E1 24246.801,E2 24246.801} C_VEL
LIN {X 0,Y 496.703,Z 363.112,A -85,B 0,C 180,E1 24246.16,E2 24246.16} C_VEL
LIN {X 0,Y 496.69,Z 363.113,A -85,B 0,C 180,E1 24242.648,E2 24242.648} C_VEL
LIN {X 0,Y 496.739,Z 363.111,A -85,B 0,C 180,E1 24239.282,E2 24239.282} C_VEL
LIN {X 0,Y 496.711,Z 363.113,A -85,B 0,C 180,E1 24235.889,E2 24235.889} C_VEL
LIN {X 0,Y 496.689,Z 363.113,A -85,B 0,C 180,E1 24232.487,E2 24232.487} C_VEL
LIN {X 0,Y 496.74,Z 363.11,A -85,B 0,C 180,E1 24229.152,E2 24229.152} C_VEL
LIN {X 0,Y 496.705,Z 363.114,A -85,B 0,C 180,E1 24225.768,E2 24225.768} C_VEL
LIN {X 0,Y 496.688,Z 363.112,A -85,B 0,C 180,E1 24222.32,E2 24222.32} C_VEL
LIN {X 0,Y 496.732,Z 363.111,A -85,B 0,C 180,E1 24218.916,E2 24218.916} C_VEL
LIN {X 0,Y 496.71,Z 363.112,A -85,B 0,C 180,E1 24215.545,E2 24215.545} C_VEL
LIN {X 0,Y 496.685,Z 363.114,A -85,B 0,C 180,E1 24212.077,E2 24212.077} C_VEL
LIN {X 0,Y 496.729,Z 363.113,A -85,B 0,C 180,E1 24208.731,E2 24208.731} C_VEL
LIN {X 0,Y 496.72,Z 363.112,A -85,B 0,C 180,E1 24205.266,E2 24205.266} C_VEL
LIN {X 0,Y 496.687,Z 363.114,A -85,B 0,C 180,E1 24201.9,E2 24201.9} C_VEL
LIN {X 0,Y 496.723,Z 363.111,A -85,B 0,C 180,E1 24198.506,E2 24198.506} C_VEL
LIN {X 0,Y 496.711,Z 363.113,A -85,B 0,C 180,E1 24195.189,E2 24195.189} C_VEL
LIN {X 0,Y 496.689,Z 363.113,A -85,B 0,C 180,E1 24191.806,E2 24191.806} C_VEL
LIN {X 0,Y 496.729,Z 363.111,A -85,B 0,C 180,E1 24188.386,E2 24188.386} C_VEL
LIN {X 0,Y 496.717,Z 363.113,A -85,B 0,C 180,E1 24184.995,E2 24184.995} C_VEL
LIN {X 0,Y 496.691,Z 363.112,A -85,B 0,C 180,E1 24181.588,E2 24181.588} C_VEL
LIN {X 0,Y 496.726,Z 363.111,A -85,B 0,C 180,E1 24178.173,E2 24178.173} C_VEL
LIN {X 0,Y 496.721,Z 363.113,A -85,B 0,C 180,E1 24174.795,E2 24174.795} C_VEL
LIN {X 0,Y 496.688,Z 363.112,A -85,B 0,C 180,E1 24171.345,E2 24171.345} C_VEL
LIN {X 0,Y 496.718,Z 363.112,A -85,B 0,C 180,E1 24167.911,E2 24167.911} C_VEL
LIN {X 0,Y 496.738,Z 363.111,A -85,B 0,C 180,E1 24164.454,E2 24164.454} C_VEL
LIN {X 0,Y 496.688,Z 363.112,A -85,B 0,C 180,E1 24161.158,E2 24161.158} C_VEL
LIN {X 0,Y 496.714,Z 363.11,A -85,B 0,C 180,E1 24157.715,E2 24157.715} C_VEL
LIN {X 0,Y 496.739,Z 363.112,A -85,B 0,C 180,E1 24154.296,E2 24154.296} C_VEL
LIN {X 0,Y 496.693,Z 363.112,A -85,B 0,C 180,E1 24150.877,E2 24150.877} C_VEL
LIN {X 0,Y 496.701,Z 363.111,A -85,B 0,C 180,E1 24147.312,E2 24147.312} C_VEL
LIN {X 0,Y 496.749,Z 363.087,A -85,B 0,C 180,E1 24143.857,E2 24143.857} C_VEL
LIN {X 0,Y 496.703,Z 363.111,A -85,B 0,C 180,E1 24140.496,E2 24140.496} C_VEL
LIN {X 0,Y 496.69,Z 363.087,A -85,B 0,C 180,E1 24136.965,E2 24136.965} C_VEL
LIN {X 0,Y 496.74,Z 363.11,A -85,B 0,C 180,E1 24133.548,E2 24133.548} C_VEL
LIN {X 0,Y 496.712,Z 363.091,A -85,B 0,C 180,E1 24130.165,E2 24130.165} C_VEL
LIN {X 0,Y 496.693,Z 363.108,A -85,B 0,C 180,E1 24126.816,E2 24126.816} C_VEL
LIN {X 0,Y 496.744,Z 363.095,A -85,B 0,C 180,E1 24123.457,E2 24123.457} C_VEL
LIN {X 0,Y 496.712,Z 363.094,A -85,B 0,C 180,E1 24119.995,E2 24119.995} C_VEL
LIN {X 0,Y 496.692,Z 363.109,A -85,B 0,C 180,E1 24116.533,E2 24116.533} C_VEL
LIN {X 0,Y 496.733,Z 363.086,A -85,B 0,C 180,E1 24113.175,E2 24113.175} C_VEL
LIN {X 0,Y 496.719,Z 363.11,A -85,B 0,C 180,E1 24109.793,E2 24109.793} C_VEL
LIN {X 0,Y 496.693,Z 363.09,A -85,B 0,C 180,E1 24106.373,E2 24106.373} C_VEL
LIN {X 0,Y 496.731,Z 363.11,A -85,B 0,C 180,E1 24102.957,E2 24102.957} C_VEL
LIN {X 0,Y 496.719,Z 363.096,A -85,B 0,C 180,E1 24099.617,E2 24099.617} C_VEL
LIN {X 0,Y 496.695,Z 363.109,A -85,B 0,C 180,E1 24096.255,E2 24096.255} C_VEL
LIN {X 0,Y 496.735,Z 363.088,A -85,B 0,C 180,E1 24092.808,E2 24092.808} C_VEL
LIN {X 0,Y 496.719,Z 363.11,A -85,B 0,C 180,E1 24089.486,E2 24089.486} C_VEL
LIN {X 0,Y 496.696,Z 363.103,A -85,B 0,C 180,E1 24086.031,E2 24086.031} C_VEL
LIN {X 0,Y 496.735,Z 363.098,A -85,B 0,C 180,E1 24082.66,E2 24082.66} C_VEL
LIN {X 0,Y 496.716,Z 363.111,A -85,B 0,C 180,E1 24079.363,E2 24079.363} C_VEL
LIN {X 0,Y 496.698,Z 363.11,A -85,B 0,C 180,E1 24075.941,E2 24075.941} C_VEL
LIN {X 0,Y 496.74,Z 363.096,A -85,B 0,C 180,E1 24072.546,E2 24072.546} C_VEL
LIN {X 0,Y 496.718,Z 363.114,A -85,B 0,C 180,E1 24069.194,E2 24069.194} C_VEL
LIN {X 0,Y 496.826,Z 363.628,A -85,B 0,C 180,E1 24068.935,E2 24068.935} C_VEL
LIN {X 0,Y 501.667,Z 380.163,A -85,B 0,C 180,E1 24066.068,E2 24066.068} C_VEL
LIN {X 0,Y 503.853,Z 388.442,A -85,B 0,C 180,E1 24064.716,E2 24064.716} C_VEL
LIN {X 0,Y 503.674,Z 393.573,A -85,B 0,C 180,E1 24064.055,E2 24064.055} C_VEL
LIN {X 0,Y 510.706,Z 420.023,A -85,B 0,C 180,E1 24063.084,E2 24063.084} C_VEL
LIN {X 0,Y 507.749,Z 647.469,A -85,B 0,C 180,E1 24059.592,E2 24059.592} C_VEL
LIN {X 0,Y 507.235,Z 664.935,A -85,B 0,C 180,E1 24059.213,E2 24059.213} C_VEL
LIN {X 0,Y 506.473,Z 684.409,A -85,B 0,C 180,E1 24058.619,E2 24058.619} C_VEL
LIN {X 0,Y 505.473,Z 703.37,A -85,B 0,C 180,E1 24057.827,E2 24057.827} C_VEL
LIN {X 0,Y 504.512,Z 719.605,A -85,B 0,C 180,E1 24056.989,E2 24056.989} C_VEL
LIN {X 0,Y 503.45,Z 735.874,A -85,B 0,C 180,E1 24055.987,E2 24055.987} C_VEL
LIN {X 0,Y 502.153,Z 754.613,A -85,B 0,C 180,E1 24054.591,E2 24054.591} C_VEL
LIN {X 0,Y 501.049,Z 769.525,A -85,B 0,C 180,E1 24053.272,E2 24053.272} C_VEL
LIN {X 0,Y 499.999,Z 784.198,A -85,B 0,C 180,E1 24051.773,E2 24051.773} C_VEL
LIN {X 0,Y 498.886,Z 799.469,A -85,B 0,C 180,E1 24049.92,E2 24049.92} C_VEL
LIN {X 0,Y 498.075,Z 811.221,A -85,B 0,C 180,E1 24048.249,E2 24048.249} C_VEL
LIN {X 0,Y 497.333,Z 823.507,A -85,B 0,C 180,E1 24046.227,E2 24046.227} C_VEL
LIN {X 0,Y 496.75,Z 834.176,A -85,B 0,C 180,E1 24044.096,E2 24044.096} C_VEL
LIN {X 0,Y 496.39,Z 842.15,A -85,B 0,C 180,E1 24042.21,E2 24042.21} C_VEL
LIN {X 0,Y 496.127,Z 850.314,A -85,B 0,C 180,E1 24039.863,E2 24039.863} C_VEL
LIN {X 0,Y 495.996,Z 856.178,A -85,B 0,C 180,E1 24037.645,E2 24037.645} C_VEL
LIN {X 0,Y 495.936,Z 860.14,A -85,B 0,C 180,E1 24035.669,E2 24035.669} C_VEL
LIN {X 0,Y 495.912,Z 863.436,A -85,B 0,C 180,E1 24033.236,E2 24033.236} C_VEL
LIN {X 0,Y 495.912,Z 864.793,A -85,B 0,C 180,E1 24030.924,E2 24030.924} C_VEL
LIN {X 0,Y 495.909,Z 864.735,A -85,B 0,C 180,E1 24028.845,E2 24028.845} C_VEL
LIN {X 0,Y 495.913,Z 863.067,A -85,B 0,C 180,E1 24026.405,E2 24026.405} C_VEL
LIN {X 0,Y 495.939,Z 859.934,A -85,B 0,C 180,E1 24024.215,E2 24024.215} C_VEL
LIN {X 0,Y 496.001,Z 855.911,A -85,B 0,C 180,E1 24022.238,E2 24022.238} C_VEL
LIN {X 0,Y 496.144,Z 849.605,A -85,B 0,C 180,E1 24019.903,E2 24019.903} C_VEL
LIN {X 0,Y 496.39,Z 842.15,A -85,B 0,C 180,E1 24017.79,E2 24017.79} C_VEL
LIN {X 0,Y 496.75,Z 834.176,A -85,B 0,C 180,E1 24015.904,E2 24015.904} C_VEL
LIN {X 0,Y 497.333,Z 823.507,A -85,B 0,C 180,E1 24013.773,E2 24013.773} C_VEL
LIN {X 0,Y 498.075,Z 811.221,A -85,B 0,C 180,E1 24011.751,E2 24011.751} C_VEL
LIN {X 0,Y 498.91,Z 799.174,A -85,B 0,C 180,E1 24010.041,E2 24010.041} C_VEL
LIN {X 0,Y 500.038,Z 783.635,A -85,B 0,C 180,E1 24008.167,E2 24008.167} C_VEL
LIN {X 0,Y 501.049,Z 769.525,A -85,B 0,C 180,E1 24006.728,E2 24006.728} C_VEL
LIN {X 0,Y 502.153,Z 754.613,A -85,B 0,C 180,E1 24005.409,E2 24005.409} C_VEL
LIN {X 0,Y 503.493,Z 735.201,A -85,B 0,C 180,E1 24003.969,E2 24003.969} C_VEL
LIN {X 0,Y 504.512,Z 719.605,A -85,B 0,C 180,E1 24003.011,E2 24003.011} C_VEL
LIN {X 0,Y 505.474,Z 703.37,A -85,B 0,C 180,E1 24002.173,E2 24002.173} C_VEL
LIN {X 0,Y 506.532,Z 682.857,A -85,B 0,C 180,E1 24001.329,E2 24001.329} C_VEL
LIN {X 0,Y 507.261,Z 664.003,A -85,B 0,C 180,E1 24000.763,E2 24000.763} C_VEL
LIN {X 0,Y 507.781,Z 646.236,A -85,B 0,C 180,E1 24000.386,E2 24000.386} C_VEL
LIN {X 0,Y 510.715,Z 419.314,A -85,B 0,C 180,E1 23996.905,E2 23996.905} C_VEL
LIN {X 0,Y 503.626,Z 393.202,A -85,B 0,C 180,E1 23995.921,E2 23995.921} C_VEL
LIN {X 0,Y 503.728,Z 387.463,A -85,B 0,C 180,E1 23995.135,E2 23995.135} C_VEL
LIN {X 0,Y 498.684,Z 369.921,A -85,B 0,C 180,E1 23992.185,E2 23992.185} C_VEL
LIN {X 0,Y 496.737,Z 363.156,A -85,B 0,C 180,E1 23990.95,E2 23990.95} C_VEL
LIN {X 0,Y 496.725,Z 363.094,A -85,B 0,C 180,E1 23987.6,E2 23987.6} C_VEL
LIN {X 0,Y 496.697,Z 363.11,A -85,B 0,C 180,E1 23984.15,E2 23984.15} C_VEL
LIN {X 0,Y 496.722,Z 363.109,A -85,B 0,C 180,E1 23980.71,E2 23980.71} C_VEL
LIN {X 0,Y 496.725,Z 363.099,A -85,B 0,C 180,E1 23977.441,E2 23977.441} C_VEL
LIN {X 0,Y 496.694,Z 363.104,A -85,B 0,C 180,E1 23974.033,E2 23974.033} C_VEL
LIN {X 0,Y 496.729,Z 363.11,A -85,B 0,C 180,E1 23970.618,E2 23970.618} C_VEL
LIN {X 0,Y 496.72,Z 363.088,A -85,B 0,C 180,E1 23967.323,E2 23967.323} C_VEL
LIN {X 0,Y 496.695,Z 363.109,A -85,B 0,C 180,E1 23963.871,E2 23963.871} C_VEL
LIN {X 0,Y 496.731,Z 363.092,A -85,B 0,C 180,E1 23960.506,E2 23960.506} C_VEL
LIN {X 0,Y 496.725,Z 363.11,A -85,B 0,C 180,E1 23957.095,E2 23957.095} C_VEL
LIN {X 0,Y 496.692,Z 363.09,A -85,B 0,C 180,E1 23953.745,E2 23953.745} C_VEL
LIN {X 0,Y 496.73,Z 363.11,A -85,B 0,C 180,E1 23950.324,E2 23950.324} C_VEL
LIN {X 0,Y 496.721,Z 363.088,A -85,B 0,C 180,E1 23946.941,E2 23946.941} C_VEL
LIN {X 0,Y 496.692,Z 363.109,A -85,B 0,C 180,E1 23943.583,E2 23943.583} C_VEL
LIN {X 0,Y 496.736,Z 363.095,A -85,B 0,C 180,E1 23940.236,E2 23940.236} C_VEL
LIN {X 0,Y 496.722,Z 363.094,A -85,B 0,C 180,E1 23936.774,E2 23936.774} C_VEL
LIN {X 0,Y 496.691,Z 363.108,A -85,B 0,C 180,E1 23933.417,E2 23933.417} C_VEL
LIN {X 0,Y 496.732,Z 363.087,A -85,B 0,C 180,E1 23930.037,E2 23930.037} C_VEL
LIN {X 0,Y 496.722,Z 363.11,A -85,B 0,C 180,E1 23926.622,E2 23926.622} C_VEL
LIN {X 0,Y 496.689,Z 363.087,A -85,B 0,C 180,E1 23923.276,E2 23923.276} C_VEL
LIN {X 0,Y 496.734,Z 363.112,A -85,B 0,C 180,E1 23919.874,E2 23919.874} C_VEL
LIN {X 0,Y 496.715,Z 363.094,A -85,B 0,C 180,E1 23916.519,E2 23916.519} C_VEL
LIN {X 0,Y 496.692,Z 363.112,A -85,B 0,C 180,E1 23913.076,E2 23913.076} C_VEL
LIN {X 0,Y 496.728,Z 363.112,A -85,B 0,C 180,E1 23909.661,E2 23909.661} C_VEL
LIN {X 0,Y 496.724,Z 363.112,A -85,B 0,C 180,E1 23906.259,E2 23906.259} C_VEL
LIN {X 0,Y 496.69,Z 363.11,A -85,B 0,C 180,E1 23902.858,E2 23902.858} C_VEL
LIN {X 0,Y 496.723,Z 363.111,A -85,B 0,C 180,E1 23899.456,E2 23899.456} C_VEL
LIN {X 0,Y 496.729,Z 363.112,A -85,B 0,C 180,E1 23896.028,E2 23896.028} C_VEL
LIN {X 0,Y 496.69,Z 363.112,A -85,B 0,C 180,E1 23892.717,E2 23892.717} C_VEL
LIN {X 0,Y 496.728,Z 363.111,A -85,B 0,C 180,E1 23889.349,E2 23889.349} C_VEL
LIN {X 0,Y 496.703,Z 363.112,A -85,B 0,C 180,E1 23886.16,E2 23886.16} C_VEL
LIN {X 0,Y 495.742,Z 363.236,A -85,B 0,C 180,E1 23885.271,E2 23885.271} C_VEL
LIN {X 0,Y 489.272,Z 364.039,A -85,B 0,C 180,E1 23882.772,E2 23882.772} C_VEL
LIN {X 0,Y 488.763,Z 364.102,A -85,B 0,C 180,E1 23882.12,E2 23882.12} C_VEL
LIN {X 0,Y 488.751,Z 364.101,A -85,B 0,C 180,E1 23878.6,E2 23878.6} C_VEL
LIN {X 0,Y 488.794,Z 364.1,A -85,B 0,C 180,E1 23875.18,E2 23875.18} C_VEL
LIN {X 0,Y 488.773,Z 364.101,A -85,B 0,C 180,E1 23871.787,E2 23871.787} C_VEL
LIN {X 0,Y 488.75,Z 364.102,A -85,B 0,C 180,E1 23868.363,E2 23868.363} C_VEL
LIN {X 0,Y 488.784,Z 364.103,A -85,B 0,C 180,E1 23864.936,E2 23864.936} C_VEL
LIN {X 0,Y 488.777,Z 364.1,A -85,B 0,C 180,E1 23861.564,E2 23861.564} C_VEL
LIN {X 0,Y 488.749,Z 364.103,A -85,B 0,C 180,E1 23858.115,E2 23858.115} C_VEL
LIN {X 0,Y 488.777,Z 364.101,A -85,B 0,C 180,E1 23854.693,E2 23854.693} C_VEL
LIN {X 0,Y 488.8,Z 364.1,A -85,B 0,C 180,E1 23851.172,E2 23851.172} C_VEL
LIN {X 0,Y 488.75,Z 364.103,A -85,B 0,C 180,E1 23847.772,E2 23847.772} C_VEL
LIN {X 0,Y 488.751,Z 364.103,A -85,B 0,C 180,E1 23844.129,E2 23844.129} C_VEL
LIN {X 0,Y 488.81,Z 364.098,A -85,B 0,C 180,E1 23840.82,E2 23840.82} C_VEL
LIN {X 0,Y 488.765,Z 364.101,A -85,B 0,C 180,E1 23837.325,E2 23837.325} C_VEL
LIN {X 0,Y 488.75,Z 364.103,A -85,B 0,C 180,E1 23833.846,E2 23833.846} C_VEL
LIN {X 0,Y 488.789,Z 364.1,A -85,B 0,C 180,E1 23830.399,E2 23830.399} C_VEL
LIN {X 0,Y 488.781,Z 364.102,A -85,B 0,C 180,E1 23826.98,E2 23826.98} C_VEL
LIN {X 0,Y 488.751,Z 364.102,A -85,B 0,C 180,E1 23823.515,E2 23823.515} C_VEL
LIN {X 0,Y 488.772,Z 364.1,A -85,B 0,C 180,E1 23820.058,E2 23820.058} C_VEL
LIN {X 0,Y 488.804,Z 364.099,A -85,B 0,C 180,E1 23816.617,E2 23816.617} C_VEL
LIN {X 0,Y 488.754,Z 364.102,A -85,B 0,C 180,E1 23813.174,E2 23813.174} C_VEL
LIN {X 0,Y 488.754,Z 364.1,A -85,B 0,C 180,E1 23809.541,E2 23809.541} C_VEL
LIN {X 0,Y 488.802,Z 364.099,A -85,B 0,C 180,E1 23806.099,E2 23806.099} C_VEL
LIN {X 0,Y 488.781,Z 364.101,A -85,B 0,C 180,E1 23802.607,E2 23802.607} C_VEL
LIN {X 0,Y 488.751,Z 364.1,A -85,B 0,C 180,E1 23799.167,E2 23799.167} C_VEL
LIN {X 0,Y 488.777,Z 364.101,A -85,B 0,C 180,E1 23795.699,E2 23795.699} C_VEL
LIN {X 0,Y 488.801,Z 364.101,A -85,B 0,C 180,E1 23792.26,E2 23792.26} C_VEL
LIN {X 0,Y 488.755,Z 364.1,A -85,B 0,C 180,E1 23788.86,E2 23788.86} C_VEL
LIN {X 0,Y 488.76,Z 364.088,A -85,B 0,C 180,E1 23785.288,E2 23785.288} C_VEL
LIN {X 0,Y 488.819,Z 364.091,A -85,B 0,C 180,E1 23781.849,E2 23781.849} C_VEL
LIN {X 0,Y 488.771,Z 364.088,A -85,B 0,C 180,E1 23778.349,E2 23778.349} C_VEL
LIN {X 0,Y 488.752,Z 364.096,A -85,B 0,C 180,E1 23774.931,E2 23774.931} C_VEL
LIN {X 0,Y 488.801,Z 364.087,A -85,B 0,C 180,E1 23771.541,E2 23771.541} C_VEL
LIN {X 0,Y 488.787,Z 364.08,A -85,B 0,C 180,E1 23767.99,E2 23767.99} C_VEL
LIN {X 0,Y 488.755,Z 364.098,A -85,B 0,C 180,E1 23764.571,E2 23764.571} C_VEL
LIN {X 0,Y 488.767,Z 364.076,A -85,B 0,C 180,E1 23761.05,E2 23761.05} C_VEL
LIN {X 0,Y 488.806,Z 364.099,A -85,B 0,C 180,E1 23757.65,E2 23757.65} C_VEL
LIN {X 0,Y 488.755,Z 364.08,A -85,B 0,C 180,E1 23754.242,E2 23754.242} C_VEL
LIN {X 0,Y 488.757,Z 364.099,A -85,B 0,C 180,E1 23750.576,E2 23750.576} C_VEL
LIN {X 0,Y 488.799,Z 364.077,A -85,B 0,C 180,E1 23747.113,E2 23747.113} C_VEL
LIN {X 0,Y 488.77,Z 364.09,A -85,B 0,C 180,E1 23743.842,E2 23743.842} C_VEL
LIN {X 0,Y 488.758,Z 364.092,A -85,B 0,C 180,E1 23740.393,E2 23740.393} C_VEL
LIN {X 0,Y 488.807,Z 364.087,A -85,B 0,C 180,E1 23736.992,E2 23736.992} C_VEL
LIN {X 0,Y 488.782,Z 364.091,A -85,B 0,C 180,E1 23733.513,E2 23733.513} C_VEL
LIN {X 0,Y 488.757,Z 364.098,A -85,B 0,C 180,E1 23730.052,E2 23730.052} C_VEL
LIN {X 0,Y 488.782,Z 364.087,A -85,B 0,C 180,E1 23726.573,E2 23726.573} C_VEL
LIN {X 0,Y 488.806,Z 364.09,A -85,B 0,C 180,E1 23723.108,E2 23723.108} C_VEL
LIN {X 0,Y 488.759,Z 364.102,A -85,B 0,C 180,E1 23719.723,E2 23719.723} C_VEL
LIN {X 0,Y 488.763,Z 364.099,A -85,B 0,C 180,E1 23716.09,E2 23716.09} C_VEL
LIN {X 0,Y 488.807,Z 364.083,A -85,B 0,C 180,E1 23712.613,E2 23712.613} C_VEL
LIN {X 0,Y 488.776,Z 364.226,A -85,B 0,C 180,E1 23709.583,E2 23709.583} C_VEL
LIN {X 0,Y 493.587,Z 380.469,A -85,B 0,C 180,E1 23706.659,E2 23706.659} C_VEL
LIN {X 0,Y 496.407,Z 391.058,A -85,B 0,C 180,E1 23704.891,E2 23704.891} C_VEL
LIN {X 0,Y 496.442,Z 393.545,A -85,B 0,C 180,E1 23704.615,E2 23704.615} C_VEL
LIN {X 0,Y 503.967,Z 421.74,A -85,B 0,C 180,E1 23703.552,E2 23703.552} C_VEL
LIN {X 0,Y 500.775,Z 647.643,A -85,B 0,C 180,E1 23700.038,E2 23700.038} C_VEL
LIN {X 0,Y 500.212,Z 665.162,A -85,B 0,C 180,E1 23699.651,E2 23699.651} C_VEL
LIN {X 0,Y 499.337,Z 685.408,A -85,B 0,C 180,E1 23699.016,E2 23699.016} C_VEL
LIN {X 0,Y 498.246,Z 704.376,A -85,B 0,C 180,E1 23698.202,E2 23698.202} C_VEL
LIN {X 0,Y 497.223,Z 720.296,A -85,B 0,C 180,E1 23697.361,E2 23697.361} C_VEL
LIN {X 0,Y 495.938,Z 738.625,A -85,B 0,C 180,E1 23696.2,E2 23696.2} C_VEL
LIN {X 0,Y 494.606,Z 755.797,A -85,B 0,C 180,E1 23694.864,E2 23694.864} C_VEL
LIN {X 0,Y 493.475,Z 769.915,A -85,B 0,C 180,E1 23693.588,E2 23693.588} C_VEL
LIN {X 0,Y 492.259,Z 785.635,A -85,B 0,C 180,E1 23691.945,E2 23691.945} C_VEL
LIN {X 0,Y 491.107,Z 800.214,A -85,B 0,C 180,E1 23690.125,E2 23690.125} C_VEL
LIN {X 0,Y 490.248,Z 811.985,A -85,B 0,C 180,E1 23688.428,E2 23688.428} C_VEL
LIN {X 0,Y 489.445,Z 824.145,A -85,B 0,C 180,E1 23686.374,E2 23686.374} C_VEL
LIN {X 0,Y 488.843,Z 834.17,A -85,B 0,C 180,E1 23684.328,E2 23684.328} C_VEL
LIN {X 0,Y 488.448,Z 842.147,A -85,B 0,C 180,E1 23682.411,E2 23682.411} C_VEL
LIN {X 0,Y 488.161,Z 849.964,A -85,B 0,C 180,E1 23680.145,E2 23680.145} C_VEL
LIN {X 0,Y 488.007,Z 855.906,A -85,B 0,C 180,E1 23677.89,E2 23677.89} C_VEL
LIN {X 0,Y 487.942,Z 859.932,A -85,B 0,C 180,E1 23675.88,E2 23675.88} C_VEL
LIN {X 0,Y 487.912,Z 863.214,A -85,B 0,C 180,E1 23673.525,E2 23673.525} C_VEL
LIN {X 0,Y 487.908,Z 864.731,A -85,B 0,C 180,E1 23671.174,E2 23671.174} C_VEL
LIN {X 0,Y 487.909,Z 864.818,A -85,B 0,C 180,E1 23669.178,E2 23669.178} C_VEL
LIN {X 0,Y 487.914,Z 863.7,A -85,B 0,C 180,E1 23667.063,E2 23667.063} C_VEL
LIN {X 0,Y 487.932,Z 860.754,A -85,B 0,C 180,E1 23664.591,E2 23664.591} C_VEL
LIN {X 0,Y 487.994,Z 856.707,A -85,B 0,C 180,E1 23662.465,E2 23662.465} C_VEL
LIN {X 0,Y 488.116,Z 851.631,A -85,B 0,C 180,E1 23660.45,E2 23660.45} C_VEL
LIN {X 0,Y 488.374,Z 844.265,A -85,B 0,C 180,E1 23658.136,E2 23658.136} C_VEL
LIN {X 0,Y 488.789,Z 835.243,A -85,B 0,C 180,E1 23655.912,E2 23655.912} C_VEL
LIN {X 0,Y 489.315,Z 825.987,A -85,B 0,C 180,E1 23653.987,E2 23653.987} C_VEL
LIN {X 0,Y 490.15,Z 813.572,A -85,B 0,C 180,E1 23651.814,E2 23651.814} C_VEL
LIN {X 0,Y 490.971,Z 802.001,A -85,B 0,C 180,E1 23650.118,E2 23650.118} C_VEL
LIN {X 0,Y 491.955,Z 789.17,A -85,B 0,C 180,E1 23648.479,E2 23648.479} C_VEL
LIN {X 0,Y 493.287,Z 772.562,A -85,B 0,C 180,E1 23646.667,E2 23646.667} C_VEL
LIN {X 0,Y 494.488,Z 757.224,A -85,B 0,C 180,E1 23645.257,E2 23645.257} C_VEL
LIN {X 0,Y 495.726,Z 741.245,A -85,B 0,C 180,E1 23643.995,E2 23643.995} C_VEL
LIN {X 0,Y 497.147,Z 721.495,A -85,B 0,C 180,E1 23642.707,E2 23642.707} C_VEL
LIN {X 0,Y 498.215,Z 704.938,A -85,B 0,C 180,E1 23641.826,E2 23641.826} C_VEL
LIN {X 0,Y 499.227,Z 687.073,A -85,B 0,C 180,E1 23641.05,E2 23641.05} C_VEL
LIN {X 0,Y 500.196,Z 665.744,A -85,B 0,C 180,E1 23640.364,E2 23640.364} C_VEL
LIN {X 0,Y 500.763,Z 648.054,A -85,B 0,C 180,E1 23639.969,E2 23639.969} C_VEL
LIN {X 0,Y 503.948,Z 423.194,A -85,B 0,C 180,E1 23636.471,E2 23636.471} C_VEL
LIN {X 0,Y 503.683,Z 419.969,A -85,B 0,C 180,E1 23636.397,E2 23636.397} C_VEL
LIN {X 0,Y 496.34,Z 392.918,A -85,B 0,C 180,E1 23635.35,E2 23635.35} C_VEL
LIN {X 0,Y 496.181,Z 389.736,A -85,B 0,C 180,E1 23634.901,E2 23634.901} C_VEL
LIN {X 0,Y 491.474,Z 373.299,A -85,B 0,C 180,E1 23632.094,E2 23632.094} C_VEL
LIN {X 0,Y 488.767,Z 364.163,A -85,B 0,C 180,E1 23630.397,E2 23630.397} C_VEL
LIN {X 0,Y 488.808,Z 364.089,A -85,B 0,C 180,E1 23627.068,E2 23627.068} C_VEL
LIN {X 0,Y 488.785,Z 364.098,A -85,B 0,C 180,E1 23623.583,E2 23623.583} C_VEL
LIN {X 0,Y 488.758,Z 364.101,A -85,B 0,C 180,E1 23620.124,E2 23620.124} C_VEL
LIN {X 0,Y 488.785,Z 364.097,A -85,B 0,C 180,E1 23616.681,E2 23616.681} C_VEL
LIN {X 0,Y 488.802,Z 364.084,A -85,B 0,C 180,E1 23613.218,E2 23613.218} C_VEL
LIN {X 0,Y 488.757,Z 364.098,A -85,B 0,C 180,E1 23609.812,E2 23609.812} C_VEL
LIN {X 0,Y 488.765,Z 364.098,A -85,B 0,C 180,E1 23606.227,E2 23606.227} C_VEL
LIN {X 0,Y 488.817,Z 364.081,A -85,B 0,C 180,E1 23602.746,E2 23602.746} C_VEL
LIN {X 0,Y 488.777,Z 364.091,A -85,B 0,C 180,E1 23599.233,E2 23599.233} C_VEL
LIN {X 0,Y 488.755,Z 364.09,A -85,B 0,C 180,E1 23595.792,E2 23595.792} C_VEL
LIN {X 0,Y 488.795,Z 364.086,A -85,B 0,C 180,E1 23592.407,E2 23592.407} C_VEL
LIN {X 0,Y 488.793,Z 364.096,A -85,B 0,C 180,E1 23588.893,E2 23588.893} C_VEL
LIN {X 0,Y 488.753,Z 364.081,A -85,B 0,C 180,E1 23585.522,E2 23585.522} C_VEL
LIN {X 0,Y 488.774,Z 364.098,A -85,B 0,C 180,E1 23581.998,E2 23581.998} C_VEL
LIN {X 0,Y 488.802,Z 364.07,A -85,B 0,C 180,E1 23578.599,E2 23578.599} C_VEL
LIN {X 0,Y 488.756,Z 364.098,A -85,B 0,C 180,E1 23575.194,E2 23575.194} C_VEL
LIN {X 0,Y 488.755,Z 364.08,A -85,B 0,C 180,E1 23571.536,E2 23571.536} C_VEL
LIN {X 0,Y 488.801,Z 364.093,A -85,B 0,C 180,E1 23568.083,E2 23568.083} C_VEL
LIN {X 0,Y 488.771,Z 364.094,A -85,B 0,C 180,E1 23564.705,E2 23564.705} C_VEL
LIN {X 0,Y 488.753,Z 364.094,A -85,B 0,C 180,E1 23561.272,E2 23561.272} C_VEL
LIN {X 0,Y 488.8,Z 364.089,A -85,B 0,C 180,E1 23557.898,E2 23557.898} C_VEL
LIN {X 0,Y 488.78,Z 364.087,A -85,B 0,C 180,E1 23554.434,E2 23554.434} C_VEL
LIN {X 0,Y 488.754,Z 364.1,A -85,B 0,C 180,E1 23551.006,E2 23551.006} C_VEL
LIN {X 0,Y 488.786,Z 364.102,A -85,B 0,C 180,E1 23547.601,E2 23547.601} C_VEL
LIN {X 0,Y 488.801,Z 364.1,A -85,B 0,C 180,E1 23544.06,E2 23544.06} C_VEL
LIN {X 0,Y 488.752,Z 364.1,A -85,B 0,C 180,E1 23540.648,E2 23540.648} C_VEL
LIN {X 0,Y 488.759,Z 364.101,A -85,B 0,C 180,E1 23537.072,E2 23537.072} C_VEL
LIN {X 0,Y 488.808,Z 364.099,A -85,B 0,C 180,E1 23533.617,E2 23533.617} C_VEL
LIN {X 0,Y 488.76,Z 364.1,A -85,B 0,C 180,E1 23530.272,E2 23530.272} C_VEL
LIN {X 0,Y 488.751,Z 364.102,A -85,B 0,C 180,E1 23526.699,E2 23526.699} C_VEL
LIN {X 0,Y 488.786,Z 364.102,A -85,B 0,C 180,E1 23523.228,E2 23523.228} C_VEL
LIN {X 0,Y 488.763,Z 364.102,A -85,B 0,C 180,E1 23522.12,E2 23522.12} C_VEL
LIN {X 0,Y 487.798,Z 364.225,A -85,B 0,C 180,E1 23521.216,E2 23521.216} C_VEL
LIN {X 0,Y 481.328,Z 365.027,A -85,B 0,C 180,E1 23518.676,E2 23518.676} C_VEL
LIN {X 0,Y 480.826,Z 365.09,A -85,B 0,C 180,E1 23518.013,E2 23518.013} C_VEL
LIN {X 0,Y 480.811,Z 365.092,A -85,B 0,C 180,E1 23514.445,E2 23514.445} C_VEL
LIN {X 0,Y 480.838,Z 365.089,A -85,B 0,C 180,E1 23510.956,E2 23510.956} C_VEL
LIN {X 0,Y 480.865,Z 365.088,A -85,B 0,C 180,E1 23507.401,E2 23507.401} C_VEL
LIN {X 0,Y 480.815,Z 365.092,A -85,B 0,C 180,E1 23503.958,E2 23503.958} C_VEL
LIN {X 0,Y 480.811,Z 365.092,A -85,B 0,C 180,E1 23500.302,E2 23500.302} C_VEL
LIN {X 0,Y 480.846,Z 365.092,A -85,B 0,C 180,E1 23496.807,E2 23496.807} C_VEL
LIN {X 0,Y 480.847,Z 365.09,A -85,B 0,C 180,E1 23493.338,E2 23493.338} C_VEL
LIN {X 0,Y 480.809,Z 365.093,A -85,B 0,C 180,E1 23489.881,E2 23489.881} C_VEL
LIN {X 0,Y 480.818,Z 365.09,A -85,B 0,C 180,E1 23486.304,E2 23486.304} C_VEL
LIN {X 0,Y 480.876,Z 365.086,A -85,B 0,C 180,E1 23482.834,E2 23482.834} C_VEL
LIN {X 0,Y 480.828,Z 365.09,A -85,B 0,C 180,E1 23479.335,E2 23479.335} C_VEL
LIN {X 0,Y 480.809,Z 365.092,A -85,B 0,C 180,E1 23475.796,E2 23475.796} C_VEL
LIN {X 0,Y 480.84,Z 365.091,A -85,B 0,C 180,E1 23472.327,E2 23472.327} C_VEL
LIN {X 0,Y 480.866,Z 365.089,A -85,B 0,C 180,E1 23468.79,E2 23468.79} C_VEL
LIN {X 0,Y 480.818,Z 365.092,A -85,B 0,C 180,E1 23465.294,E2 23465.294} C_VEL
LIN {X 0,Y 480.814,Z 365.09,A -85,B 0,C 180,E1 23461.698,E2 23461.698} C_VEL
LIN {X 0,Y 480.855,Z 365.088,A -85,B 0,C 180,E1 23458.244,E2 23458.244} C_VEL
LIN {X 0,Y 480.854,Z 365.089,A -85,B 0,C 180,E1 23454.687,E2 23454.687} C_VEL
LIN {X 0,Y 480.813,Z 365.09,A -85,B 0,C 180,E1 23451.23,E2 23451.23} C_VEL
LIN {X 0,Y 480.818,Z 365.09,A -85,B 0,C 180,E1 23447.568,E2 23447.568} C_VEL
LIN {X 0,Y 480.868,Z 365.088,A -85,B 0,C 180,E1 23444.14,E2 23444.14} C_VEL
LIN {X 0,Y 480.838,Z 365.089,A -85,B 0,C 180,E1 23440.627,E2 23440.627} C_VEL
LIN {X 0,Y 480.813,Z 365.088,A -85,B 0,C 180,E1 23437.209,E2 23437.209} C_VEL
LIN {X 0,Y 480.845,Z 365.09,A -85,B 0,C 180,E1 23433.715,E2 23433.715} C_VEL
LIN {X 0,Y 480.863,Z 365.09,A -85,B 0,C 180,E1 23430.203,E2 23430.203} C_VEL
LIN {X 0,Y 480.817,Z 365.09,A -85,B 0,C 180,E1 23426.816,E2 23426.816} C_VEL
LIN {X 0,Y 480.817,Z 365.075,A -85,B 0,C 180,E1 23423.135,E2 23423.135} C_VEL
LIN {X 0,Y 480.863,Z 365.082,A -85,B 0,C 180,E1 23419.678,E2 23419.678} C_VEL
LIN {X 0,Y 480.846,Z 365.063,A -85,B 0,C 180,E1 23416.128,E2 23416.128} C_VEL
LIN {X 0,Y 480.813,Z 365.089,A -85,B 0,C 180,E1 23412.728,E2 23412.728} C_VEL
LIN {X 0,Y 480.832,Z 365.061,A -85,B 0,C 180,E1 23409.208,E2 23409.208} C_VEL
LIN {X 0,Y 480.86,Z 365.087,A -85,B 0,C 180,E1 23405.842,E2 23405.842} C_VEL
LIN {X 0,Y 480.816,Z 365.068,A -85,B 0,C 180,E1 23402.378,E2 23402.378} C_VEL
LIN {X 0,Y 480.818,Z 365.087,A -85,B 0,C 180,E1 23398.684,E2 23398.684} C_VEL
LIN {X 0,Y 480.856,Z 365.069,A -85,B 0,C 180,E1 23395.224,E2 23395.224} C_VEL
LIN {X 0,Y 480.842,Z 365.073,A -85,B 0,C 180,E1 23391.794,E2 23391.794} C_VEL
LIN {X 0,Y 480.817,Z 365.085,A -85,B 0,C 180,E1 23388.354,E2 23388.354} C_VEL
LIN {X 0,Y 480.835,Z 365.07,A -85,B 0,C 180,E1 23384.807,E2 23384.807} C_VEL
LIN {X 0,Y 480.873,Z 365.084,A -85,B 0,C 180,E1 23381.321,E2 23381.321} C_VEL
LIN {X 0,Y 480.821,Z 365.068,A -85,B 0,C 180,E1 23377.886,E2 23377.886} C_VEL
LIN {X 0,Y 480.823,Z 365.086,A -85,B 0,C 180,E1 23374.368,E2 23374.368} C_VEL
LIN {X 0,Y 480.867,Z 365.072,A -85,B 0,C 180,E1 23370.882,E2 23370.882} C_VEL
LIN {X 0,Y 480.845,Z 365.079,A -85,B 0,C 180,E1 23367.411,E2 23367.411} C_VEL
LIN {X 0,Y 480.818,Z 365.09,A -85,B 0,C 180,E1 23363.946,E2 23363.946} C_VEL
LIN {X 0,Y 480.845,Z 365.09,A -85,B 0,C 180,E1 23360.481,E2 23360.481} C_VEL
LIN {X 0,Y 480.87,Z 365.087,A -85,B 0,C 180,E1 23356.997,E2 23356.997} C_VEL
LIN {X 0,Y 480.828,Z 365.094,A -85,B 0,C 180,E1 23353.467,E2 23353.467} C_VEL
LIN {X 0,Y 480.852,Z 365.227,A -85,B 0,C 180,E1 23350.154,E2 23350.154} C_VEL
LIN {X 0,Y 485.683,Z 381.29,A -85,B 0,C 180,E1 23347.181,E2 23347.181} C_VEL
LIN {X 0,Y 488.951,Z 392.973,A -85,B 0,C 180,E1 23345.23,E2 23345.23} C_VEL
LIN {X 0,Y 496.368,Z 419.42,A -85,B 0,C 180,E1 23344.17,E2 23344.17} C_VEL
LIN {X 0,Y 497.26,Z 423.822,A -85,B 0,C 180,E1 23344.026,E2 23344.026} C_VEL
LIN {X 0,Y 493.829,Z 647.919,A -85,B 0,C 180,E1 23340.495,E2 23340.495} C_VEL
LIN {X 0,Y 493.211,Z 665.667,A -85,B 0,C 180,E1 23340.094,E2 23340.094} C_VEL
LIN {X 0,Y 492.145,Z 687.404,A -85,B 0,C 180,E1 23339.382,E2 23339.382} C_VEL
LIN {X 0,Y 491.089,Z 704.61,A -85,B 0,C 180,E1 23338.625,E2 23338.625} C_VEL
LIN {X 0,Y 489.937,Z 721.254,A -85,B 0,C 180,E1 23337.729,E2 23337.729} C_VEL
LIN {X 0,Y 488.414,Z 740.824,A -85,B 0,C 180,E1 23336.439,E2 23336.439} C_VEL
LIN {X 0,Y 487.134,Z 756.269,A -85,B 0,C 180,E1 23335.207,E2 23335.207} C_VEL
LIN {X 0,Y 485.918,Z 770.305,A -85,B 0,C 180,E1 23333.913,E2 23333.913} C_VEL
LIN {X 0,Y 484.554,Z 786.42,A -85,B 0,C 180,E1 23332.185,E2 23332.185} C_VEL
LIN {X 0,Y 483.388,Z 800.098,A -85,B 0,C 180,E1 23330.442,E2 23330.442} C_VEL
LIN {X 0,Y 482.446,Z 811.901,A -85,B 0,C 180,E1 23328.712,E2 23328.712} C_VEL
LIN {X 0,Y 481.546,Z 824.637,A -85,B 0,C 180,E1 23326.526,E2 23326.526} C_VEL
LIN {X 0,Y 480.944,Z 834.158,A -85,B 0,C 180,E1 23324.569,E2 23324.569} C_VEL
LIN {X 0,Y 480.512,Z 842.144,A -85,B 0,C 180,E1 23322.62,E2 23322.62} C_VEL
LIN {X 0,Y 480.191,Z 849.967,A -85,B 0,C 180,E1 23320.315,E2 23320.315} C_VEL
LIN {X 0,Y 480.016,Z 855.901,A -85,B 0,C 180,E1 23318.022,E2 23318.022} C_VEL
LIN {X 0,Y 479.946,Z 859.93,A -85,B 0,C 180,E1 23315.979,E2 23315.979} C_VEL
LIN {X 0,Y 479.915,Z 863.134,A -85,B 0,C 180,E1 23313.652,E2 23313.652} C_VEL
LIN {X 0,Y 479.908,Z 864.727,A -85,B 0,C 180,E1 23311.194,E2 23311.194} C_VEL
LIN {X 0,Y 479.909,Z 864.814,A -85,B 0,C 180,E1 23309.164,E2 23309.164} C_VEL
LIN {X 0,Y 479.913,Z 863.695,A -85,B 0,C 180,E1 23307.014,E2 23307.014} C_VEL
LIN {X 0,Y 479.935,Z 860.752,A -85,B 0,C 180,E1 23304.501,E2 23304.501} C_VEL
LIN {X 0,Y 480.004,Z 856.702,A -85,B 0,C 180,E1 23302.339,E2 23302.339} C_VEL
LIN {X 0,Y 480.137,Z 851.625,A -85,B 0,C 180,E1 23300.289,E2 23300.289} C_VEL
LIN {X 0,Y 480.415,Z 844.45,A -85,B 0,C 180,E1 23297.988,E2 23297.988} C_VEL
LIN {X 0,Y 480.854,Z 835.774,A -85,B 0,C 180,E1 23295.797,E2 23295.797} C_VEL
LIN {X 0,Y 481.369,Z 827.12,A -85,B 0,C 180,E1 23293.964,E2 23293.964} C_VEL
LIN {X 0,Y 482.126,Z 816.339,A -85,B 0,C 180,E1 23292.001,E2 23292.001} C_VEL
LIN {X 0,Y 483.178,Z 802.651,A -85,B 0,C 180,E1 23289.91,E2 23289.91} C_VEL
LIN {X 0,Y 484.188,Z 790.431,A -85,B 0,C 180,E1 23288.307,E2 23288.307} C_VEL
LIN {X 0,Y 485.413,Z 776.398,A -85,B 0,C 180,E1 23286.705,E2 23286.705} C_VEL
LIN {X 0,Y 486.868,Z 759.341,A -85,B 0,C 180,E1 23285.058,E2 23285.058} C_VEL
LIN {X 0,Y 488.085,Z 744.866,A -85,B 0,C 180,E1 23283.869,E2 23283.869} C_VEL
LIN {X 0,Y 489.336,Z 729.183,A -85,B 0,C 180,E1 23282.762,E2 23282.762} C_VEL
LIN {X 0,Y 490.813,Z 709.124,A -85,B 0,C 180,E1 23281.598,E2 23281.598} C_VEL
LIN {X 0,Y 491.872,Z 691.869,A -85,B 0,C 180,E1 23280.801,E2 23280.801} C_VEL
LIN {X 0,Y 492.799,Z 674.705,A -85,B 0,C 180,E1 23280.172,E2 23280.172} C_VEL
LIN {X 0,Y 493.705,Z 653.105,A -85,B 0,C 180,E1 23279.603,E2 23279.603} C_VEL
LIN {X 0,Y 494.494,Z 607.904,A -85,B 0,C 180,E1 23278.864,E2 23278.864} C_VEL
LIN {X 0,Y 497.167,Z 422.422,A -85,B 0,C 180,E1 23275.943,E2 23275.943} C_VEL
LIN {X 0,Y 488.985,Z 393.063,A -85,B 0,C 180,E1 23274.777,E2 23274.777} C_VEL
LIN {X 0,Y 487.168,Z 386.778,A -85,B 0,C 180,E1 23273.767,E2 23273.767} C_VEL
LIN {X 0,Y 482.416,Z 370.257,A -85,B 0,C 180,E1 23270.822,E2 23270.822} C_VEL
LIN {X 0,Y 480.845,Z 365.169,A -85,B 0,C 180,E1 23269.826,E2 23269.826} C_VEL
LIN {X 0,Y 480.822,Z 365.094,A -85,B 0,C 180,E1 23266.341,E2 23266.341} C_VEL
LIN {X 0,Y 480.855,Z 365.086,A -85,B 0,C 180,E1 23262.842,E2 23262.842} C_VEL
LIN {X 0,Y 480.86,Z 365.09,A -85,B 0,C 180,E1 23259.363,E2 23259.363} C_VEL
LIN {X 0,Y 480.82,Z 365.09,A -85,B 0,C 180,E1 23255.906,E2 23255.906} C_VEL
LIN {X 0,Y 480.826,Z 365.086,A -85,B 0,C 180,E1 23252.308,E2 23252.308} C_VEL
LIN {X 0,Y 480.877,Z 365.065,A -85,B 0,C 180,E1 23248.845,E2 23248.845} C_VEL
LIN {X 0,Y 480.837,Z 365.086,A -85,B 0,C 180,E1 23245.367,E2 23245.367} C_VEL
LIN {X 0,Y 480.815,Z 365.068,A -85,B 0,C 180,E1 23241.857,E2 23241.857} C_VEL
LIN {X 0,Y 480.85,Z 365.09,A -85,B 0,C 180,E1 23238.429,E2 23238.429} C_VEL
LIN {X 0,Y 480.858,Z 365.063,A -85,B 0,C 180,E1 23234.946,E2 23234.946} C_VEL
LIN {X 0,Y 480.818,Z 365.085,A -85,B 0,C 180,E1 23231.52,E2 23231.52} C_VEL
LIN {X 0,Y 480.821,Z 365.072,A -85,B 0,C 180,E1 23227.893,E2 23227.893} C_VEL
LIN {X 0,Y 480.873,Z 365.071,A -85,B 0,C 180,E1 23224.537,E2 23224.537} C_VEL
LIN {X 0,Y 480.828,Z 365.087,A -85,B 0,C 180,E1 23221.077,E2 23221.077} C_VEL
LIN {X 0,Y 480.814,Z 365.07,A -85,B 0,C 180,E1 23217.502,E2 23217.502} C_VEL
LIN {X 0,Y 480.848,Z 365.086,A -85,B 0,C 180,E1 23214.038,E2 23214.038} C_VEL
LIN {X 0,Y 480.843,Z 365.059,A -85,B 0,C 180,E1 23210.672,E2 23210.672} C_VEL
LIN {X 0,Y 480.814,Z 365.089,A -85,B 0,C 180,E1 23207.229,E2 23207.229} C_VEL
LIN {X 0,Y 480.831,Z 365.062,A -85,B 0,C 180,E1 23203.703,E2 23203.703} C_VEL
LIN {X 0,Y 480.874,Z 365.083,A -85,B 0,C 180,E1 23200.196,E2 23200.196} C_VEL
LIN {X 0,Y 480.822,Z 365.073,A -85,B 0,C 180,E1 23196.735,E2 23196.735} C_VEL
LIN {X 0,Y 480.815,Z 365.09,A -85,B 0,C 180,E1 23193.136,E2 23193.136} C_VEL
LIN {X 0,Y 480.848,Z 365.09,A -85,B 0,C 180,E1 23189.645,E2 23189.645} C_VEL
LIN {X 0,Y 480.859,Z 365.089,A -85,B 0,C 180,E1 23186.143,E2 23186.143} C_VEL
LIN {X 0,Y 480.818,Z 365.088,A -85,B 0,C 180,E1 23182.621,E2 23182.621} C_VEL
LIN {X 0,Y 480.816,Z 365.09,A -85,B 0,C 180,E1 23179.011,E2 23179.011} C_VEL
LIN {X 0,Y 480.858,Z 365.089,A -85,B 0,C 180,E1 23175.526,E2 23175.526} C_VEL
LIN {X 0,Y 480.843,Z 365.089,A -85,B 0,C 180,E1 23172.032,E2 23172.032} C_VEL
LIN {X 0,Y 480.81,Z 365.09,A -85,B 0,C 180,E1 23168.578,E2 23168.578} C_VEL
LIN {X 0,Y 480.828,Z 365.091,A -85,B 0,C 180,E1 23165.023,E2 23165.023} C_VEL
LIN {X 0,Y 480.875,Z 365.087,A -85,B 0,C 180,E1 23161.533,E2 23161.533} C_VEL
LIN {X 0,Y 480.817,Z 365.09,A -85,B 0,C 180,E1 23158.166,E2 23158.166} C_VEL
LIN {X 0,Y 480.826,Z 365.09,A -85,B 0,C 180,E1 23158.013,E2 23158.013} C_VEL
LIN {X 0,Y 479.866,Z 365.215,A -85,B 0,C 180,E1 23157.095,E2 23157.095} C_VEL
LIN {X 0,Y 473.395,Z 366.019,A -85,B 0,C 180,E1 23154.513,E2 23154.513} C_VEL
LIN {X 0,Y 472.896,Z 366.08,A -85,B 0,C 180,E1 23153.839,E2 23153.839} C_VEL
LIN {X 0,Y 472.872,Z 366.079,A -85,B 0,C 180,E1 23150.418,E2 23150.418} C_VEL
LIN {X 0,Y 472.907,Z 366.078,A -85,B 0,C 180,E1 23146.963,E2 23146.963} C_VEL
LIN {X 0,Y 472.915,Z 366.077,A -85,B 0,C 180,E1 23143.448,E2 23143.448} C_VEL
LIN {X 0,Y 472.873,Z 366.081,A -85,B 0,C 180,E1 23139.984,E2 23139.984} C_VEL
LIN {X 0,Y 472.875,Z 366.081,A -85,B 0,C 180,E1 23136.312,E2 23136.312} C_VEL
LIN {X 0,Y 472.91,Z 366.078,A -85,B 0,C 180,E1 23132.787,E2 23132.787} C_VEL
LIN {X 0,Y 472.907,Z 366.078,A -85,B 0,C 180,E1 23129.273,E2 23129.273} C_VEL
LIN {X 0,Y 472.872,Z 366.079,A -85,B 0,C 180,E1 23125.756,E2 23125.756} C_VEL
LIN {X 0,Y 472.874,Z 366.082,A -85,B 0,C 180,E1 23122.101,E2 23122.101} C_VEL
LIN {X 0,Y 472.92,Z 366.079,A -85,B 0,C 180,E1 23118.661,E2 23118.661} C_VEL
LIN {X 0,Y 472.895,Z 366.081,A -85,B 0,C 180,E1 23115.177,E2 23115.177} C_VEL
LIN {X 0,Y 472.873,Z 366.081,A -85,B 0,C 180,E1 23111.637,E2 23111.637} C_VEL
LIN {X 0,Y 472.882,Z 366.08,A -85,B 0,C 180,E1 23108.023,E2 23108.023} C_VEL
LIN {X 0,Y 472.928,Z 366.076,A -85,B 0,C 180,E1 23104.502,E2 23104.502} C_VEL
LIN {X 0,Y 472.89,Z 366.078,A -85,B 0,C 180,E1 23101.042,E2 23101.042} C_VEL
LIN {X 0,Y 472.873,Z 366.08,A -85,B 0,C 180,E1 23097.512,E2 23097.512} C_VEL
LIN {X 0,Y 472.899,Z 366.08,A -85,B 0,C 180,E1 23094.002,E2 23094.002} C_VEL
LIN {X 0,Y 472.931,Z 366.077,A -85,B 0,C 180,E1 23090.48,E2 23090.48} C_VEL
LIN {X 0,Y 472.884,Z 366.08,A -85,B 0,C 180,E1 23086.927,E2 23086.927} C_VEL
LIN {X 0,Y 472.875,Z 366.08,A -85,B 0,C 180,E1 23083.336,E2 23083.336} C_VEL
LIN {X 0,Y 472.906,Z 366.078,A -85,B 0,C 180,E1 23079.828,E2 23079.828} C_VEL
LIN {X 0,Y 472.924,Z 366.078,A -85,B 0,C 180,E1 23076.288,E2 23076.288} C_VEL
LIN {X 0,Y 472.882,Z 366.08,A -85,B 0,C 180,E1 23072.762,E2 23072.762} C_VEL
LIN {X 0,Y 472.878,Z 366.078,A -85,B 0,C 180,E1 23069.164,E2 23069.164} C_VEL
LIN {X 0,Y 472.912,Z 366.064,A -85,B 0,C 180,E1 23065.677,E2 23065.677} C_VEL
LIN {X 0,Y 472.921,Z 366.065,A -85,B 0,C 180,E1 23062.099,E2 23062.099} C_VEL
LIN {X 0,Y 472.879,Z 366.07,A -85,B 0,C 180,E1 23058.612,E2 23058.612} C_VEL
LIN {X 0,Y 472.875,Z 366.074,A -85,B 0,C 180,E1 23054.925,E2 23054.925} C_VEL
LIN {X 0,Y 472.914,Z 366.063,A -85,B 0,C 180,E1 23051.457,E2 23051.457} C_VEL
LIN {X 0,Y 472.919,Z 366.056,A -85,B 0,C 180,E1 23047.893,E2 23047.893} C_VEL
LIN {X 0,Y 472.882,Z 366.076,A -85,B 0,C 180,E1 23044.36,E2 23044.36} C_VEL
LIN {X 0,Y 472.875,Z 366.055,A -85,B 0,C 180,E1 23040.722,E2 23040.722} C_VEL
LIN {X 0,Y 472.926,Z 366.075,A -85,B 0,C 180,E1 23037.329,E2 23037.329} C_VEL
LIN {X 0,Y 472.904,Z 366.047,A -85,B 0,C 180,E1 23033.805,E2 23033.805} C_VEL
LIN {X 0,Y 472.878,Z 366.077,A -85,B 0,C 180,E1 23030.38,E2 23030.38} C_VEL
LIN {X 0,Y 472.891,Z 366.053,A -85,B 0,C 180,E1 23026.796,E2 23026.796} C_VEL
LIN {X 0,Y 472.929,Z 366.068,A -85,B 0,C 180,E1 23023.412,E2 23023.412} C_VEL
LIN {X 0,Y 472.883,Z 366.066,A -85,B 0,C 180,E1 23019.965,E2 23019.965} C_VEL
LIN {X 0,Y 472.88,Z 366.076,A -85,B 0,C 180,E1 23016.278,E2 23016.278} C_VEL
LIN {X 0,Y 472.918,Z 366.051,A -85,B 0,C 180,E1 23012.824,E2 23012.824} C_VEL
LIN {X 0,Y 472.913,Z 366.077,A -85,B 0,C 180,E1 23009.363,E2 23009.363} C_VEL
LIN {X 0,Y 472.879,Z 366.069,A -85,B 0,C 180,E1 23005.919,E2 23005.919} C_VEL
LIN {X 0,Y 472.891,Z 366.064,A -85,B 0,C 180,E1 23002.331,E2 23002.331} C_VEL
LIN {X 0,Y 472.944,Z 366.063,A -85,B 0,C 180,E1 22998.816,E2 22998.816} C_VEL
LIN {X 0,Y 472.903,Z 366.069,A -85,B 0,C 180,E1 22995.243,E2 22995.243} C_VEL
LIN {X 0,Y 472.877,Z 366.039,A -85,B 0,C 180,E1 22991.718,E2 22991.718} C_VEL
LIN {X 0,Y 472.98,Z 366.32,A -85,B 0,C 180,E1 22990.717,E2 22990.717} C_VEL
LIN {X 0,Y 478.122,Z 383.472,A -85,B 0,C 180,E1 22987.483,E2 22987.483} C_VEL
LIN {X 0,Y 480.68,Z 392.597,A -85,B 0,C 180,E1 22985.931,E2 22985.931} C_VEL
LIN {X 0,Y 483.642,Z 398.881,A -85,B 0,C 180,E1 22985.557,E2 22985.557} C_VEL
LIN {X 0,Y 490.597,Z 425.27,A -85,B 0,C 180,E1 22984.524,E2 22984.524} C_VEL
LIN {X 0,Y 486.918,Z 648.093,A -85,B 0,C 180,E1 22980.966,E2 22980.966} C_VEL
LIN {X 0,Y 486.242,Z 666.122,A -85,B 0,C 180,E1 22980.551,E2 22980.551} C_VEL
LIN {X 0,Y 485.078,Z 687.908,A -85,B 0,C 180,E1 22979.819,E2 22979.819} C_VEL
LIN {X 0,Y 483.94,Z 705.144,A -85,B 0,C 180,E1 22979.046,E2 22979.046} C_VEL
LIN {X 0,Y 482.683,Z 722.079,A -85,B 0,C 180,E1 22978.115,E2 22978.115} C_VEL
LIN {X 0,Y 481.046,Z 741.391,A -85,B 0,C 180,E1 22976.809,E2 22976.809} C_VEL
LIN {X 0,Y 479.679,Z 756.74,A -85,B 0,C 180,E1 22975.561,E2 22975.561} C_VEL
LIN {X 0,Y 478.291,Z 771.677,A -85,B 0,C 180,E1 22974.151,E2 22974.151} C_VEL
LIN {X 0,Y 476.752,Z 788.183,A -85,B 0,C 180,E1 22972.308,E2 22972.308} C_VEL
LIN {X 0,Y 475.624,Z 800.622,A -85,B 0,C 180,E1 22970.681,E2 22970.681} C_VEL
LIN {X 0,Y 474.62,Z 812.294,A -85,B 0,C 180,E1 22968.93,E2 22968.93} C_VEL
LIN {X 0,Y 473.639,Z 825.015,A -85,B 0,C 180,E1 22966.684,E2 22966.684} C_VEL
LIN {X 0,Y 472.998,Z 834.46,A -85,B 0,C 180,E1 22964.694,E2 22964.694} C_VEL
LIN {X 0,Y 472.546,Z 842.468,A -85,B 0,C 180,E1 22962.712,E2 22962.712} C_VEL
LIN {X 0,Y 472.177,Z 850.936,A -85,B 0,C 180,E1 22960.122,E2 22960.122} C_VEL
LIN {X 0,Y 472.021,Z 856.163,A -85,B 0,C 180,E1 22958.036,E2 22958.036} C_VEL
LIN {X 0,Y 471.948,Z 860.133,A -85,B 0,C 180,E1 22955.958,E2 22955.958} C_VEL
LIN {X 0,Y 471.913,Z 863.333,A -85,B 0,C 180,E1 22953.523,E2 22953.523} C_VEL
LIN {X 0,Y 471.911,Z 864.753,A -85,B 0,C 180,E1 22951.093,E2 22951.093} C_VEL
LIN {X 0,Y 471.912,Z 864.781,A -85,B 0,C 180,E1 22949.029,E2 22949.029} C_VEL
LIN {X 0,Y 471.913,Z 863.603,A -85,B 0,C 180,E1 22946.842,E2 22946.842} C_VEL
LIN {X 0,Y 471.942,Z 860.544,A -85,B 0,C 180,E1 22944.286,E2 22944.286} C_VEL
LIN {X 0,Y 472.015,Z 856.697,A -85,B 0,C 180,E1 22942.209,E2 22942.209} C_VEL
LIN {X 0,Y 472.149,Z 851.94,A -85,B 0,C 180,E1 22940.247,E2 22940.247} C_VEL
LIN {X 0,Y 472.421,Z 845.147,A -85,B 0,C 180,E1 22938.03,E2 22938.03} C_VEL
LIN {X 0,Y 472.903,Z 836.09,A -85,B 0,C 180,E1 22935.678,E2 22935.678} C_VEL
LIN {X 0,Y 473.454,Z 827.499,A -85,B 0,C 180,E1 22933.814,E2 22933.814} C_VEL
LIN {X 0,Y 474.199,Z 817.505,A -85,B 0,C 180,E1 22931.944,E2 22931.944} C_VEL
LIN {X 0,Y 475.368,Z 803.602,A -85,B 0,C 180,E1 22929.737,E2 22929.737} C_VEL
LIN {X 0,Y 476.479,Z 791.078,A -85,B 0,C 180,E1 22928.053,E2 22928.053} C_VEL
LIN {X 0,Y 477.722,Z 777.787,A -85,B 0,C 180,E1 22926.497,E2 22926.497} C_VEL
LIN {X 0,Y 479.356,Z 760.305,A -85,B 0,C 180,E1 22924.752,E2 22924.752} C_VEL
LIN {X 0,Y 480.763,Z 744.624,A -85,B 0,C 180,E1 22923.44,E2 22923.44} C_VEL
LIN {X 0,Y 482.114,Z 728.942,A -85,B 0,C 180,E1 22922.32,E2 22922.32} C_VEL
LIN {X 0,Y 483.699,Z 708.889,A -85,B 0,C 180,E1 22921.141,E2 22921.141} C_VEL
LIN {X 0,Y 484.835,Z 691.63,A -85,B 0,C 180,E1 22920.335,E2 22920.335} C_VEL
LIN {X 0,Y 485.84,Z 674.353,A -85,B 0,C 180,E1 22919.697,E2 22919.697} C_VEL
LIN {X 0,Y 486.8,Z 652.574,A -85,B 0,C 180,E1 22919.119,E2 22919.119} C_VEL
LIN {X 0,Y 487.688,Z 604.696,A -85,B 0,C 180,E1 22918.329,E2 22918.329} C_VEL
LIN {X 0,Y 490.527,Z 424.275,A -85,B 0,C 180,E1 22915.453,E2 22915.453} C_VEL
LIN {X 0,Y 482.96,Z 397.023,A -85,B 0,C 180,E1 22914.352,E2 22914.352} C_VEL
LIN {X 0,Y 480.554,Z 392.259,A -85,B 0,C 180,E1 22914.037,E2 22914.037} C_VEL
LIN {X 0,Y 475.987,Z 376.267,A -85,B 0,C 180,E1 22911.202,E2 22911.202} C_VEL
LIN {X 0,Y 472.956,Z 366.152,A -85,B 0,C 180,E1 22909.215,E2 22909.215} C_VEL
LIN {X 0,Y 472.908,Z 366.073,A -85,B 0,C 180,E1 22905.589,E2 22905.589} C_VEL
LIN {X 0,Y 472.881,Z 366.071,A -85,B 0,C 180,E1 22902.087,E2 22902.087} C_VEL
LIN {X 0,Y 472.893,Z 366.068,A -85,B 0,C 180,E1 22898.53,E2 22898.53} C_VEL
LIN {X 0,Y 472.934,Z 366.071,A -85,B 0,C 180,E1 22894.959,E2 22894.959} C_VEL
LIN {X 0,Y 472.898,Z 366.075,A -85,B 0,C 180,E1 22891.486,E2 22891.486} C_VEL
LIN {X 0,Y 472.878,Z 366.051,A -85,B 0,C 180,E1 22887.999,E2 22887.999} C_VEL
LIN {X 0,Y 472.909,Z 366.077,A -85,B 0,C 180,E1 22884.485,E2 22884.485} C_VEL
LIN {X 0,Y 472.929,Z 366.047,A -85,B 0,C 180,E1 22880.938,E2 22880.938} C_VEL
LIN {X 0,Y 472.883,Z 366.078,A -85,B 0,C 180,E1 22877.476,E2 22877.476} C_VEL
LIN {X 0,Y 472.876,Z 366.051,A -85,B 0,C 180,E1 22873.828,E2 22873.828} C_VEL
LIN {X 0,Y 472.916,Z 366.077,A -85,B 0,C 180,E1 22870.357,E2 22870.357} C_VEL
LIN {X 0,Y 472.916,Z 366.046,A -85,B 0,C 180,E1 22866.804,E2 22866.804} C_VEL
LIN {X 0,Y 472.881,Z 366.076,A -85,B 0,C 180,E1 22863.278,E2 22863.278} C_VEL
LIN {X 0,Y 472.876,Z 366.058,A -85,B 0,C 180,E1 22859.642,E2 22859.642} C_VEL
LIN {X 0,Y 472.915,Z 366.068,A -85,B 0,C 180,E1 22856.126,E2 22856.126} C_VEL
LIN {X 0,Y 472.921,Z 366.063,A -85,B 0,C 180,E1 22852.541,E2 22852.541} C_VEL
LIN {X 0,Y 472.879,Z 366.063,A -85,B 0,C 180,E1 22849.036,E2 22849.036} C_VEL
LIN {X 0,Y 472.877,Z 366.074,A -85,B 0,C 180,E1 22845.433,E2 22845.433} C_VEL
LIN {X 0,Y 472.924,Z 366.05,A -85,B 0,C 180,E1 22842.028,E2 22842.028} C_VEL
LIN {X 0,Y 472.906,Z 366.078,A -85,B 0,C 180,E1 22838.475,E2 22838.475} C_VEL
LIN {X 0,Y 472.874,Z 366.064,A -85,B 0,C 180,E1 22834.991,E2 22834.991} C_VEL
LIN {X 0,Y 472.893,Z 366.079,A -85,B 0,C 180,E1 22831.464,E2 22831.464} C_VEL
LIN {X 0,Y 472.935,Z 366.078,A -85,B 0,C 180,E1 22827.968,E2 22827.968} C_VEL
LIN {X 0,Y 472.888,Z 366.08,A -85,B 0,C 180,E1 22824.457,E2 22824.457} C_VEL
LIN {X 0,Y 472.876,Z 366.078,A -85,B 0,C 180,E1 22820.893,E2 22820.893} C_VEL
LIN {X 0,Y 472.901,Z 366.079,A -85,B 0,C 180,E1 22817.371,E2 22817.371} C_VEL
LIN {X 0,Y 472.924,Z 366.076,A -85,B 0,C 180,E1 22813.879,E2 22813.879} C_VEL
LIN {X 0,Y 472.878,Z 366.078,A -85,B 0,C 180,E1 22810.444,E2 22810.444} C_VEL
LIN {X 0,Y 472.875,Z 366.08,A -85,B 0,C 180,E1 22806.753,E2 22806.753} C_VEL
LIN {X 0,Y 472.907,Z 366.08,A -85,B 0,C 180,E1 22803.201,E2 22803.201} C_VEL
LIN {X 0,Y 472.923,Z 366.077,A -85,B 0,C 180,E1 22799.651,E2 22799.651} C_VEL
LIN {X 0,Y 472.876,Z 366.081,A -85,B 0,C 180,E1 22796.225,E2 22796.225} C_VEL
LIN {X 0,Y 472.896,Z 366.08,A -85,B 0,C 180,E1 22793.839,E2 22793.839} C_VEL
LIN {X 0,Y 472.065,Z 366.185,A -85,B 0,C 180,E1 22792.971,E2 22792.971} C_VEL
LIN {X 0,Y 468.006,Z 366.69,A -85,B 0,C 180,E1 22791.41,E2 22791.41} C_VEL
LIN {X 0,Y 465.286,Z 367.025,A -85,B 0,C 180,E1 22790.144,E2 22790.144} C_VEL
LIN {X 0,Y 464.972,Z 367.067,A -85,B 0,C 180,E1 22789.595,E2 22789.595} C_VEL
LIN {X 0,Y 464.938,Z 367.071,A -85,B 0,C 180,E1 22786.03,E2 22786.03} C_VEL
LIN {X 0,Y 464.937,Z 367.068,A -85,B 0,C 180,E1 22782.418,E2 22782.418} C_VEL
LIN {X 0,Y 464.973,Z 367.066,A -85,B 0,C 180,E1 22778.906,E2 22778.906} C_VEL
LIN {X 0,Y 464.964,Z 367.067,A -85,B 0,C 180,E1 22775.429,E2 22775.429} C_VEL
LIN {X 0,Y 464.934,Z 367.07,A -85,B 0,C 180,E1 22771.849,E2 22771.849} C_VEL
LIN {X 0,Y 464.934,Z 367.07,A -85,B 0,C 180,E1 22768.151,E2 22768.151} C_VEL
LIN {X 0,Y 464.964,Z 367.067,A -85,B 0,C 180,E1 22764.571,E2 22764.571} C_VEL
LIN {X 0,Y 464.973,Z 367.066,A -85,B 0,C 180,E1 22761.094,E2 22761.094} C_VEL
LIN {X 0,Y 464.937,Z 367.068,A -85,B 0,C 180,E1 22757.582,E2 22757.582} C_VEL
LIN {X 0,Y 464.935,Z 367.071,A -85,B 0,C 180,E1 22753.894,E2 22753.894} C_VEL
LIN {X 0,Y 464.966,Z 367.067,A -85,B 0,C 180,E1 22750.341,E2 22750.341} C_VEL
LIN {X 0,Y 464.981,Z 367.067,A -85,B 0,C 180,E1 22746.828,E2 22746.828} C_VEL
LIN {X 0,Y 464.94,Z 367.07,A -85,B 0,C 180,E1 22743.292,E2 22743.292} C_VEL
LIN {X 0,Y 464.934,Z 367.068,A -85,B 0,C 180,E1 22739.645,E2 22739.645} C_VEL
LIN {X 0,Y 464.971,Z 367.067,A -85,B 0,C 180,E1 22736.156,E2 22736.156} C_VEL
LIN {X 0,Y 464.99,Z 367.065,A -85,B 0,C 180,E1 22732.495,E2 22732.495} C_VEL
LIN {X 0,Y 464.944,Z 367.068,A -85,B 0,C 180,E1 22728.997,E2 22728.997} C_VEL
LIN {X 0,Y 464.937,Z 367.069,A -85,B 0,C 180,E1 22725.372,E2 22725.372} C_VEL
LIN {X 0,Y 464.959,Z 367.068,A -85,B 0,C 180,E1 22721.797,E2 22721.797} C_VEL
LIN {X 0,Y 464.995,Z 367.066,A -85,B 0,C 180,E1 22718.253,E2 22718.253} C_VEL
LIN {X 0,Y 464.946,Z 367.069,A -85,B 0,C 180,E1 22714.732,E2 22714.732} C_VEL
LIN {X 0,Y 464.938,Z 367.068,A -85,B 0,C 180,E1 22711.143,E2 22711.143} C_VEL
LIN {X 0,Y 464.967,Z 367.068,A -85,B 0,C 180,E1 22707.634,E2 22707.634} C_VEL
LIN {X 0,Y 464.99,Z 367.036,A -85,B 0,C 180,E1 22703.971,E2 22703.971} C_VEL
